// ---- POUs/Block/Cabines/Servomoteur_V1.TcPOU
FUNCTION_BLOCK Servomoteur_V1
VAR_INPUT
	Enable:					BOOL;	(*Mise en route du bloc de fonction*)
	Type_Consigne:			BOOL;	 (*Choix du type de pilotage du registre / 1 = ANA / 0 = TOR*)
	Mode_Vidange:			BOOL; 	(*Mode de vidange / 1=Mode vidange / 0= Mode alimentation douche, Douchette, Lavabo, etc...*)
	Cons_Pos_Dem:			REAL; 	(*Consigne position registre demandé (Venant de la régulation) / en %*)
	Cmd_Ouv_Dem:			BOOL; 	(*Commande ouverture registre demandé (Venant de la régulation) / 1 = Ouverture*)
	Info_Mes_Pos:			REAL; 	(*Info mesure position registre (recopie EAN) / en %*)
	Presence_Fdc:			INT; 	(*Mot de présence des fin de course / 0 = Pas de fin de course / 1 = Fin de course Ouvert / 2 = Fin de course Fermé / 3 = Les 2 fin de course*)
	Info_Fdc_Ouvert:			BOOL; 	(*Info fin de course ouvert (recopie ETOR) / 1 = Ouvert*)
	Info_Fdc_Ferme:			BOOL; 	(*Info fin de course fermé (recopi ETOR) / 1 = Fermé*)
	Secu_Niveau_Haut:		BOOL; 	(*Sécurité du niveau haut / 0 = Niveau haut actif*)
	Control_Discrodance:		BOOL;	 (*Autorisation de marche des alarmes / 1 = Alarme autorisé*)
	Hyst_Al_Discord:			REAL;	 (*Hystéresis pour le défaut discordance en type ANA*)
	Tempo_Discord_TOR:		TIME; 	(*Temporisation du défaut discordance en type TOR*)
	EF_Forcage:				BOOL;	 (*Enable forçage du registre / 1= Autorisé*)
	F_STOR_Registre: 		BOOL;	 (*Forçage du registre pour le mode TOR / 1= Forcé*)
	F_SAN_Registre:			REAL; 	(*Forçage du registre pour le mode ANA / en %*)
	Defaut_Alim_Eau:			BOOL;	(*Défaut sur l'alimentation d'eau*)
	E_Cmd_Rearmement:		BOOL;	(*Commande de réarmement*)
	In_SCL_In_MIN_REAL: REAL;
	In_SCL_In_MAX_REAL: REAL;
	In_SCL_Out_MIN_REAL: REAL;
	In_SCL_Out_MAX_REAL: REAL;
END_VAR
VAR_OUTPUT
	SAN_Cons_Registre:		INT; (*Consigne a appliqué au registre ANA (pour SAN) / en %*)
	STOR_Cmd_Ouv_Registre: BOOL; (*Commande a appliqué au registre TOR (pour STOR) / 1 = Ouverture*)
	Def_Discordance_ANA:BOOL;
	Def_Discordance_Ouverture:BOOL;
	Def_Discordance_Fermeture: BOOL;
END_VAR
VAR
	Cons_Registre:			REAL;
	iCons_Registre:			INT;
	Cmd_Registre:			BOOL;
	SCL_ANA: 				SCL;
	TON_1:					TON;
	TON_2:					TON;
	TON_3:					TON;
	TON_4:					TON;
	TON_5:					TON;
	TON_6:					TON;
	RS_1:					RS;
	RS_2:					RS;
	Calcul_1: REAL;
	Calcul_2: REAL;
END_VAR

IF(Enable)
	THEN
	(*======================Gestion de la Consigne===================================*)
	IF(Type_Consigne)
		THEN			(* Gestion consigne pour un registre ANA *)
		Cmd_Registre := FALSE;
		IF(EF_Forcage)
			THEN
				Cons_Registre := F_SAN_Registre;
			ELSE
				Cons_Registre := Cons_Pos_Dem;
		END_IF;
	ELSE				 (* Gestion consigne pour un registre TOR *)
		Cons_Registre := 0.0;
		IF(EF_Forcage)
			THEN
				Cmd_Registre := F_STOR_Registre;
			ELSE
				Cmd_Registre := Cmd_Ouv_Dem;
		END_IF
	END_IF;
	
	(*======================Gestion de la sortie Analogique==============================*)
	iCons_Registre := REAL_TO_INT(Cons_Registre); (*Convertion de la consigne analogique*)
	SCL_ANA(
		IN_INT:= iCons_Registre,
		LIM_MIN_IN_REAL:= In_SCL_In_MIN_REAL,
		LIM_MAX_IN_REAL:= In_SCL_In_MAX_REAL,
		LIM_MIN_OUT_REAL:= In_SCL_Out_MIN_REAL,(*0V*)
		LIM_MAX_OUT_REAL:= In_SCL_Out_MAX_REAL,(*10V*)
		OUT_INT=> SAN_Cons_Registre);
	
	(*======================Gestion de la sortie TOR====================================*)
	IF( Mode_Vidange)
		THEN (*Gestion de la STOR en fonction du mode de vidange*)
		IF(Secu_Niveau_Haut)
			THEN
				STOR_Cmd_Ouv_Registre := TRUE;
			ELSE
				STOR_Cmd_Ouv_Registre := Cmd_Registre;
		END_IF;
	ELSE (*Gestion de la STOR en fonction du mode alimentation*)
		IF(Secu_Niveau_Haut)
			THEN
				STOR_Cmd_Ouv_Registre := FALSE;
			ELSE
				STOR_Cmd_Ouv_Registre := Cmd_Registre AND NOT Defaut_Alim_Eau;
		END_IF;
	END_IF;
	
	(*======================Gestion du défaut de discordance============================*)
	IF(Control_Discrodance)
		THEN		(*Lors du contrôle de discordance*)
			IF(Type_Consigne)
				THEN		(* Alarme discordance pour registre SAN *)
					Calcul_1 := (Cons_Registre - Hyst_Al_Discord) ;
					Calcul_2 := (Cons_Registre + Hyst_Al_Discord) ;
					TON_1(IN := ((Calcul_1 > Info_Mes_Pos) OR (Calcul_2 < Info_Mes_Pos)),PT := Tempo_Discord_TOR);
					Def_Discordance_ANA:= TON_1.Q;
			ELSE			(* Alarme discordance pour registre STOR *)
				CASE Presence_Fdc OF
					0	:	(*Mode pas de fin de course*)
							Def_Discordance_Ouverture := FALSE;
							Def_Discordance_Fermeture := FALSE;
					1	:	(*Mode Fdc ouverture uniquement*)
							TON_2(IN := ( STOR_Cmd_Ouv_Registre AND NOT Info_Fdc_Ouvert ), PT := Tempo_Discord_TOR);
							Def_Discordance_Ouverture:= TON_2.Q;
							Def_Discordance_Fermeture := FALSE;
					2	:	(*Mode Fdc fermeture uniquement*)
							TON_3(IN := ( NOT STOR_Cmd_Ouv_Registre AND NOT Info_Fdc_Ferme ), PT := Tempo_Discord_TOR);
							Def_Discordance_Fermeture:= TON_3.Q;
							Def_Discordance_Ouverture := FALSE;
					3	:	(*Mode Fdc ouverture et fermeture*)
							TON_4(IN := ((STOR_Cmd_Ouv_Registre AND NOT Info_Fdc_Ouvert)),PT := Tempo_Discord_TOR);
							TON_5(IN := ((NOT STOR_Cmd_Ouv_Registre AND NOT Info_Fdc_Ferme )),PT := Tempo_Discord_TOR);
							TON_6(IN := (Info_Fdc_Ouvert AND Info_Fdc_Ferme) ,PT := Tempo_Discord_TOR);
							RS_1(SET:= TON_4.Q, RESET1:= Info_Fdc_Ouvert OR E_Cmd_Rearmement);
							RS_2(SET:= TON_5.Q, RESET1:= Info_Fdc_Ferme OR E_Cmd_Rearmement);
							Def_Discordance_Ouverture:= RS_1.Q1 OR TON_6.Q;
							Def_Discordance_Fermeture:= RS_2.Q1 OR TON_6.Q;
	
					ELSE  (*Si Presence_Fdc > à 3*)
					Def_Discordance_Ouverture := FALSE;
					Def_Discordance_Fermeture := FALSE;
				END_CASE;
			END_IF;
		ELSE		(* Si contrôle d'alarme discordance désactivé *)
			Def_Discordance_ANA := FALSE;
			Def_Discordance_Ouverture := FALSE;
			Def_Discordance_Fermeture := FALSE;
	END_IF;
	ELSE
			SAN_Cons_Registre := 0;
			STOR_Cmd_Ouv_Registre := FALSE;
			Def_Discordance_ANA := FALSE;
			Def_Discordance_Ouverture := FALSE;
			Def_Discordance_Fermeture := FALSE;
END_IF;

END_FUNCTION_BLOCK

// ---- POUs/p_Com_Modbus_RS485.TcPOU
PROGRAM p_Com_Modbus_RS485
VAR
	//Gestion de la com avec la passerelle LED
	Com_LED: Com485_Dalcnet;
	Lecture_Dimmer 	:INT;
	Lecture_Rouge 	:INT;
	Lecture_Vert 	:INT;
	Lecture_Bleu 	:INT;
	Lecture_Blanc 	:INT;
	LED_Com_Ok		:BOOL;
	LED_Com_Error	:BOOL;
	LED_Etape		:INT;
	
	//Gestion de la com avec GVL_RegTROX.Reg_Souf_GD_FCVT01
	FCVT01_Com_Ok		:BOOL;
	FCVT01_Com_Error	:BOOL;
	FCVT01_Etape		:INT;
	FCVT01_ConsAppli	:INT;
	
	//Gestion de la com avec GVL_RegTROX.Com_RegSouf_PD_FCVT02
	FCVT02_Com_Ok		:BOOL;
	FCVT02_Com_Error	:BOOL;
	FCVT02_Etape		:INT;
	FCVT02_ConsAppli	:INT;
	
	//Gestion de la com avec GVL_RegTROX.Com_RegSouf_Cabine_FCVT03
	FCVT03_Com_Ok		:BOOL;
	FCVT03_Com_Error	:BOOL;
	FCVT03_Etape		:INT;
	FCVT03_ConsAppli	:INT;
	
	//Gestion de la com avec GVL_RegTROX.Com_Reg_Bypass_FCVT04
	FCVT04_Com_Ok		:BOOL;
	FCVT04_Com_Error	:BOOL;
	FCVT04_Etape		:INT;
	FCVT04_ConsAppli	:INT;
	
	//Gestion de la com avec GVL_RegTROX.Com_RegSouf_CabGD_FCVT05
	FCVT05_Com_Ok		:BOOL;
	FCVT05_Com_Error	:BOOL;
	FCVT05_Etape		:INT;
	FCVT05_ConsAppli	:INT;
	
	//Gestion de la com avec GVL_RegTROX.Com_RegSouf_CabPD_FCVT06
	FCVT06_Com_Ok		:BOOL;
	FCVT06_Com_Error	:BOOL;
	FCVT06_Etape		:INT;
	FCVT06_ConsAppli	:INT;
	
	//Gestion de la com avec GVL_RegTROX.Com_RegRep_FCVT07
	FCVT07_Com_Ok		:BOOL;
	FCVT07_Com_Error	:BOOL;
	FCVT07_Etape		:INT;
	FCVT07_ConsAppli	:INT;
	
	Start_2: BOOL;
	Start_3: BOOL;
	Start_4: BOOL;
	Start_41: BOOL;
	Start_5: BOOL;
	Start_6: BOOL;
	Start_61: BOOL;
	Start_7: BOOL;
	Start_8: BOOL;
	Start_9: BOOL;
	FirstCycle: BOOL := TRUE;
	F_TRIG_0: F_TRIG;
	cpt: INT;
	CTU_Cpt: CTU;
	Cons_Cpt: WORD := 4;
	TOF_0: TOF;
	test: BOOL;
	
	//Gestion des forçages
	EF_FCVT01		:BOOL;
	F_FCVT01		:REAL;
	EF_FCVT02		:BOOL;
	F_FCVT02		:REAL;
	EF_FCVT03		:BOOL;
	F_FCVT03		:REAL;
	EF_FCVT04		:BOOL;
	F_FCVT04		:REAL;
	EF_FCVT05		:BOOL;
	F_FCVT05		:REAL;
	EF_FCVT06		:BOOL;
	F_FCVT06		:REAL;
	EF_FCVT07		:BOOL;
	F_FCVT07		:REAL;
END_VAR
VAR // added by the converter: edge detectors and wires of the graphical bodies
    _w1 : BOOL;
END_VAR

_w1 := Start_4 OR Start_6 OR Start_9;
Com_LED(
    Adresse_RS485 := 1,
    Start_Chenillard := _w1,
    In_Dimmer_Cabine := Cde_Dimmer_Cabine,
    In_Rouge_Cabine := Cde_Rouge_Cabine,
    In_Vert_Cabine := Cde_Vert_Cabine,
    In_Bleu_Cabine := Cde_Bleu_Cabine,
    In_Blanc_Cabine := Cde_Blanc_Cabine); // Com485_Dalcnet
LED_Com_Ok := Com_LED.Com_Ok;
LED_Com_Error := Com_LED.Com_Error;
LED_Etape := Com_LED.etape;
Defaut_Com_Dalcnet := Com_LED.Defaut_Com;
Lecture_Dimmer := Com_LED.Out_Dimmer_Cabine;
Lecture_Rouge := Com_LED.Out_Rouge_Cabine;
Lecture_Vert := Com_LED.Out_Vert_Cabine;
Lecture_Bleu := Com_LED.Out_Bleu_Cabine;
Lecture_Blanc := Com_LED.Out_Blanc_Cabine;
CTU_Cpt(CU := _w1, RESET := Start_8, PV := Cons_Cpt); // CTU
Cpt := CTU_Cpt.CV;
Start_2 := SEL(CTU_Cpt.CV = 1, false, Com_LED.Next_Chenillard);
Start_41 := SEL(CTU_Cpt.CV = 2, false, Com_LED.Next_Chenillard);
Start_61 := SEL(CTU_Cpt.CV = 3, false, Com_LED.Next_Chenillard);
GVL_RegTROX.Com_RegSouf_GD_FCVT01(
    Adresse_RS485 := 2,
    rEcriture_Cons_Deb := GVL_RegTROX.ConsAppliDeb_RegSouf_GD_FCVT01,
    rEcriture_Cons_Max := GVL_RegTROX.ConsMax_FCVT01,
    rEcriture_Cons_Min := GVL_RegTROX.ConsMin_FCVT01,
    Ecriture_ls_m3h := 1,
    Ecr_Interface_Mode := 1,
    Etat_Ma_Ventil := TRUE,
    TOL_Defaut_Discord := 250.0,
    Start_Chenillard := Start_2,
    EF_Forcage := EF_FCVT01,
    E_Forcage := F_FCVT01); // Com485_RegTROX
FCVT01_Com_Ok := GVL_RegTROX.Com_RegSouf_GD_FCVT01.Com_Ok;
FCVT01_Com_Error := GVL_RegTROX.Com_RegSouf_GD_FCVT01.Com_Error;
GVL_RegTROX.RegSouf_GD_FCVT01.Info_Mess_Pos := GVL_RegTROX.Com_RegSouf_GD_FCVT01.MES_Pos;
GVL_RegTROX.MES_RegSouf_GD_FCVT01.Mesure_EAN := GVL_RegTROX.Com_RegSouf_GD_FCVT01.rDebit_Relative;
FCVT01_ConsAppli := GVL_RegTROX.Com_RegSouf_GD_FCVT01.Lec_Cons_Appli;
FCVT01_Etape := GVL_RegTROX.Com_RegSouf_GD_FCVT01.etape;
GVL_RegTROX.RegSouf_GD_FCVT01_DefCom := GVL_RegTROX.Com_RegSouf_GD_FCVT01.Defaut_Com;
GVL_RegTROX.RegSouf_GD_FCVT01_Def_DiscordDeb := GVL_RegTROX.Com_RegSouf_GD_FCVT01.Defaut_Discord_Debit;
Start_3 := GVL_RegTROX.Com_RegSouf_GD_FCVT01.Next_Chenillard;
GVL_RegTROX.Com_RegSouf_PD_FCVT02(
    Adresse_RS485 := 3,
    rEcriture_Cons_Deb := GVL_RegTROX.ConsAppliDeb_RegSouf_PD_FCVT02,
    rEcriture_Cons_Max := GVL_RegTROX.ConsMax_FCVT02,
    rEcriture_Cons_Min := GVL_RegTROX.ConsMin_FCVT02,
    Ecriture_ls_m3h := 1,
    Ecr_Interface_Mode := 1,
    Etat_Ma_Ventil := TRUE,
    TOL_Defaut_Discord := 40.0,
    Start_Chenillard := Start_3,
    EF_Forcage := EF_FCVT02,
    E_Forcage := F_FCVT02); // Com485_RegTROX
FCVT02_Com_Ok := GVL_RegTROX.Com_RegSouf_PD_FCVT02.Com_Ok;
FCVT02_Com_Error := GVL_RegTROX.Com_RegSouf_PD_FCVT02.Com_Error;
GVL_RegTROX.RegSouf_PD_FCVT02.Info_Mess_Pos := GVL_RegTROX.Com_RegSouf_PD_FCVT02.MES_Pos;
GVL_RegTROX.MES_RegSouf_PD_FCVT02.Mesure_EAN := GVL_RegTROX.Com_RegSouf_PD_FCVT02.rDebit_Relative;
FCVT02_ConsAppli := GVL_RegTROX.Com_RegSouf_PD_FCVT02.Lec_Cons_Appli;
FCVT02_Etape := GVL_RegTROX.Com_RegSouf_PD_FCVT02.etape;
GVL_RegTROX.RegSouf_PD_FCVT02_DefCom := GVL_RegTROX.Com_RegSouf_PD_FCVT02.Defaut_Com;
GVL_RegTROX.RegSouf_PD_FCVT02_Def_DiscordDeb := GVL_RegTROX.Com_RegSouf_PD_FCVT02.Defaut_Discord_Debit;
Start_4 := GVL_RegTROX.Com_RegSouf_PD_FCVT02.Next_Chenillard;
GVL_RegTROX.Com_RegSouf_Cabine_FCVT03(
    Adresse_RS485 := 4,
    rEcriture_Cons_Deb := GVL_RegTROX.ConsAppliDeb_RegSouf_Cabine_FCVT03,
    rEcriture_Cons_Max := GVL_RegTROX.ConsMax_FCVT03,
    rEcriture_Cons_Min := GVL_RegTROX.ConsMin_FCVT03,
    Ecriture_ls_m3h := 1,
    Ecr_Interface_Mode := 1,
    Etat_Ma_Ventil := TRUE,
    TOL_Defaut_Discord := 1020.0,
    Start_Chenillard := Start_41,
    EF_Forcage := EF_FCVT03,
    E_Forcage := F_FCVT03); // Com485_RegTROX
FCVT03_Com_Ok := GVL_RegTROX.Com_RegSouf_Cabine_FCVT03.Com_Ok;
FCVT03_Com_Error := GVL_RegTROX.Com_RegSouf_Cabine_FCVT03.Com_Error;
GVL_RegTROX.RegSouf_Cabine_FCVT03.Info_Mess_Pos := GVL_RegTROX.Com_RegSouf_Cabine_FCVT03.MES_Pos;
GVL_RegTROX.MES_RegSouf_Cabine_FCVT03.Mesure_EAN := GVL_RegTROX.Com_RegSouf_Cabine_FCVT03.rDebit_Relative;
FCVT03_ConsAppli := GVL_RegTROX.Com_RegSouf_Cabine_FCVT03.Lec_Cons_Appli;
FCVT03_Etape := GVL_RegTROX.Com_RegSouf_Cabine_FCVT03.etape;
GVL_RegTROX.RegSouf_Cabine_FCVT03_DefCom := GVL_RegTROX.Com_RegSouf_Cabine_FCVT03.Defaut_Com;
GVL_RegTROX.RegSouf_Cabine_FCVT03_Def_DiscordDeb := GVL_RegTROX.Com_RegSouf_Cabine_FCVT03.Defaut_Discord_Debit;
Start_5 := GVL_RegTROX.Com_RegSouf_Cabine_FCVT03.Next_Chenillard;
GVL_RegTROX.Com_Reg_Bypass_FCVT04(
    Adresse_RS485 := 5,
    rEcriture_Cons_Deb := GVL_RegTROX.ConsAppliDeb_Reg_Bypass_FCVT04,
    rEcriture_Cons_Max := GVL_RegTROX.ConsMax_FCVT04,
    rEcriture_Cons_Min := GVL_RegTROX.ConsMin_FCVT04,
    Ecriture_ls_m3h := 1,
    Ecr_Interface_Mode := 1,
    Etat_Ma_Ventil := TRUE,
    TOL_Defaut_Discord := 150.0,
    Start_Chenillard := Start_5,
    EF_Forcage := EF_FCVT04,
    E_Forcage := F_FCVT04); // Com485_RegTROX
FCVT04_Com_Ok := GVL_RegTROX.Com_Reg_Bypass_FCVT04.Com_Ok;
FCVT04_Com_Error := GVL_RegTROX.Com_Reg_Bypass_FCVT04.Com_Error;
GVL_RegTROX.RegBypass_FCVT04.Info_Mess_Pos := GVL_RegTROX.Com_Reg_Bypass_FCVT04.MES_Pos;
GVL_RegTROX.MES_RegBypass_FCVT04.Mesure_EAN := GVL_RegTROX.Com_Reg_Bypass_FCVT04.rDebit_Relative;
FCVT04_ConsAppli := GVL_RegTROX.Com_Reg_Bypass_FCVT04.Lec_Cons_Appli;
FCVT04_Etape := GVL_RegTROX.Com_Reg_Bypass_FCVT04.etape;
GVL_RegTROX.Reg_Bypass_FCVT04_DefCom := GVL_RegTROX.Com_Reg_Bypass_FCVT04.Defaut_Com;
GVL_RegTROX.Reg_Bypass_FCVT04_Def_DiscordDeb := GVL_RegTROX.Com_Reg_Bypass_FCVT04.Defaut_Discord_Debit;
Start_6 := GVL_RegTROX.Com_Reg_Bypass_FCVT04.Next_Chenillard;
GVL_RegTROX.Com_RegSouf_CabGD_FCVT05(
    Adresse_RS485 := 6,
    rEcriture_Cons_Deb := GVL_RegTROX.ConsAppliDeb_RegSouf_CabGD_FCVT05,
    rEcriture_Cons_Max := GVL_RegTROX.ConsMax_FCVT05,
    rEcriture_Cons_Min := GVL_RegTROX.ConsMin_FCVT05,
    Ecriture_ls_m3h := 1,
    Ecr_Interface_Mode := 1,
    Etat_Ma_Ventil := TRUE,
    TOL_Defaut_Discord := 250.0,
    Start_Chenillard := Start_61,
    EF_Forcage := EF_FCVT05,
    E_Forcage := F_FCVT05); // Com485_RegTROX
FCVT05_Com_Ok := GVL_RegTROX.Com_RegSouf_CabGD_FCVT05.Com_Ok;
FCVT05_Com_Error := GVL_RegTROX.Com_RegSouf_CabGD_FCVT05.Com_Error;
GVL_RegTROX.RegSouf_CabGD_FCVT05.Info_Mess_Pos := GVL_RegTROX.Com_RegSouf_CabGD_FCVT05.MES_Pos;
GVL_RegTROX.MES_RegSouf_CabGD_FCVT05.Mesure_EAN := GVL_RegTROX.Com_RegSouf_CabGD_FCVT05.rDebit_Relative;
FCVT05_ConsAppli := GVL_RegTROX.Com_RegSouf_CabGD_FCVT05.Lec_Cons_Appli;
FCVT05_Etape := GVL_RegTROX.Com_RegSouf_CabGD_FCVT05.etape;
GVL_RegTROX.RegSouf_CabGD_FCVT05_DefCom := GVL_RegTROX.Com_RegSouf_CabGD_FCVT05.Defaut_Com;
GVL_RegTROX.RegSouf_CabGD_FCVT05_Def_DiscordDeb := GVL_RegTROX.Com_RegSouf_CabGD_FCVT05.Defaut_Discord_Debit;
Start_7 := GVL_RegTROX.Com_RegSouf_CabGD_FCVT05.Next_Chenillard;
GVL_RegTROX.Com_RegSouf_CabPD_FCVT06(
    Adresse_RS485 := 7,
    rEcriture_Cons_Deb := GVL_RegTROX.ConsAppliDeb_RegSouf_CabPD_FCVT06,
    rEcriture_Cons_Max := GVL_RegTROX.ConsMax_FCVT06,
    rEcriture_Cons_Min := GVL_RegTROX.ConsMin_FCVT06,
    Ecriture_ls_m3h := 1,
    Ecr_Interface_Mode := 1,
    Etat_Ma_Ventil := TRUE,
    TOL_Defaut_Discord := 50.0,
    Start_Chenillard := Start_7,
    EF_Forcage := EF_FCVT06,
    E_Forcage := F_FCVT06); // Com485_RegTROX
FCVT06_Com_Ok := GVL_RegTROX.Com_RegSouf_CabPD_FCVT06.Com_Ok;
FCVT06_Com_Error := GVL_RegTROX.Com_RegSouf_CabPD_FCVT06.Com_Error;
GVL_RegTROX.RegSouf_CabPD_FCVT06.Info_Mess_Pos := GVL_RegTROX.Com_RegSouf_CabPD_FCVT06.MES_Pos;
GVL_RegTROX.MES_RegSouf_CabPD_FCVT06.Mesure_EAN := GVL_RegTROX.Com_RegSouf_CabPD_FCVT06.rDebit_Relative;
FCVT06_ConsAppli := GVL_RegTROX.Com_RegSouf_CabPD_FCVT06.Lec_Cons_Appli;
FCVT06_Etape := GVL_RegTROX.Com_RegSouf_CabPD_FCVT06.etape;
GVL_RegTROX.RegSouf_CabPD_FCVT06_DefCom := GVL_RegTROX.Com_RegSouf_CabPD_FCVT06.Defaut_Com;
GVL_RegTROX.RegSouf_CabPD_FCVT06_Def_DiscordDeb := GVL_RegTROX.Com_RegSouf_CabPD_FCVT06.Defaut_Discord_Debit;
Start_8 := GVL_RegTROX.Com_RegSouf_CabPD_FCVT06.Next_Chenillard;
GVL_RegTROX.Com_RegRep_FCVT07(
    Adresse_RS485 := 8,
    rEcriture_Cons_Deb := GVL_RegTROX.ConsAppliDeb_RegRep_FCVT07,
    rEcriture_Cons_Max := GVL_RegTROX.ConsMax_FCVT07,
    rEcriture_Cons_Min := GVL_RegTROX.ConsMin_FCVT07,
    Ecriture_ls_m3h := 1,
    Ecr_Interface_Mode := 1,
    Etat_Ma_Ventil := TRUE,
    TOL_Defaut_Discord := 1020.0,
    Start_Chenillard := Start_8,
    EF_Forcage := EF_FCVT07,
    E_Forcage := F_FCVT07); // Com485_RegTROX
FCVT07_Com_Ok := GVL_RegTROX.Com_RegRep_FCVT07.Com_Ok;
FCVT07_Com_Error := GVL_RegTROX.Com_RegRep_FCVT07.Com_Error;
GVL_RegTROX.RegRep_FCVT07.Info_Mess_Pos := GVL_RegTROX.Com_RegRep_FCVT07.MES_Pos;
GVL_RegTROX.MES_RegRep_FCVT07.Mesure_EAN := GVL_RegTROX.Com_RegRep_FCVT07.rDebit_Relative;
FCVT07_ConsAppli := GVL_RegTROX.Com_RegRep_FCVT07.Lec_Cons_Appli;
FCVT07_Etape := GVL_RegTROX.Com_RegRep_FCVT07.etape;
GVL_RegTROX.RegRep_FCVT07_DefCom := GVL_RegTROX.Com_RegRep_FCVT07.Defaut_Com;
GVL_RegTROX.RegRep_FCVT07_Def_DiscordDeb := GVL_RegTROX.Com_RegRep_FCVT07.Defaut_Discord_Debit;
F_TRIG_0(CLK := FirstCycle OR test); // F_TRIG
Start_9 := GVL_RegTROX.Com_RegRep_FCVT07.Next_Chenillard OR F_TRIG_0.Q;
TOF_0(IN := Start_2, PT := T#5m); // TOF
test := TOF_0.Q;
FirstCycle := FALSE;

END_PROGRAM

// ---- POUs/Block/Cabines/Com485_Dalcnet.TcPOU
FUNCTION_BLOCK Com485_Dalcnet
VAR_INPUT
	Adresse_RS485		:BYTE;
	Start_Chenillard	: BOOL;
	In_Dimmer_Cabine	:INT;
	In_Rouge_Cabine		:INT;
	In_Vert_Cabine		:INT;
	In_Bleu_Cabine		:INT;
	In_Blanc_Cabine		:INT;
END_VAR
VAR_OUTPUT
	Com_Ok 				: BOOL;
	Com_Error 			: BOOL;
	etape				: INT := 0;
	Defaut_Com			: BOOL;
	Next_Chenillard		: BOOL;
	Out_Dimmer_Cabine	:INT;
	Out_Rouge_Cabine	:INT;
	Out_Vert_Cabine		:INT;
	Out_Bleu_Cabine		:INT;
	Out_Blanc_Cabine	:INT;
END_VAR
VAR
	Last_Error				: MODBUS_ERRORS;
	ValeursEcrites_Dalcnet 	: ARRAY[0..5] OF INT;
	ValeursLues_Dalcnet 	: ARRAY[0..5] OF INT;
	Chgt_Ecr_Cons_Dalcnet	: BOOL;
	F_TRIG_1				: F_TRIG;
	F_TRIG_2				: F_TRIG;
	TON_1					: TON;
	TON_2					: TON;
	R_TRIG_Start			: R_TRIG;
END_VAR

(*Gestion de l'ecriture*)
ValeursEcrites_Dalcnet[0] 	:= In_Dimmer_Cabine;
ValeursEcrites_Dalcnet[1] 	:= In_Rouge_Cabine;
ValeursEcrites_Dalcnet[2] 	:= In_Vert_Cabine;
ValeursEcrites_Dalcnet[3] 	:= In_Bleu_Cabine;
ValeursEcrites_Dalcnet[4] 	:= In_Blanc_Cabine;
(*Recopie des consignes du Dalcnet*)
Out_Dimmer_Cabine 			:= ValeursLues_Dalcnet[0];
Out_Rouge_Cabine 			:= ValeursLues_Dalcnet[1];
Out_Vert_Cabine 			:= ValeursLues_Dalcnet[2];
Out_Bleu_Cabine 			:= ValeursLues_Dalcnet[3];
Out_Blanc_Cabine 			:= ValeursLues_Dalcnet[4];

(*Changement de consigne pour l'ecriture Modbus*)
IF((Out_Rouge_Cabine <> In_Rouge_Cabine) OR (Out_Vert_Cabine <> In_Vert_Cabine) OR (Out_Bleu_Cabine <> In_Bleu_Cabine) OR (Out_Blanc_Cabine <> In_Blanc_Cabine))
	THEN
	Chgt_Ecr_Cons_Dalcnet := TRUE;
	ELSE
	Chgt_Ecr_Cons_Dalcnet := FALSE;
END_IF;

(**********************************************Gestion sécurité anti-blocage*)
(*En cas de blocage de la variable etape à 0*)
TON_1(IN:=(etape = 1) , PT:= T#3S);
IF (TON_1.Q) THEN etape := 3; END_IF;

(*En cas de blocage de la variable etape à 3*)
TON_2(IN:=(etape = 3) , PT:= T#3S);
IF (TON_2.Q) THEN etape := 0; END_IF;

(**********************************************Lecture/ecriture modbus*)
CASE etape OF
	0: (*Etape Attente*)
		R_TRIG_Start(CLK:= Start_Chenillard);
		IF (R_TRIG_Start.Q)
			THEN
			etape := etape + 1;
		END_IF;
		Next_Chenillard := FALSE;
	(*Lecture dalcnet*)
	1:	MB.ReadRegs(	Execute := NOT MB.BUSY,
						UnitID := Adresse_RS485,
						Quantity := 6,								(* Lecture de 6 mots *)
						MBAddr := 16#0,							(*A partir de l'adresse 0*)
						cbLength := SIZEOF(ValeursLues_Dalcnet),
						pMemoryAddr := ADR(ValeursLues_Dalcnet),
						Timeout := T#5000MS);
		F_TRIG_1(CLK:= MB.BUSY);
		IF(F_TRIG_1.Q)
			THEN
			etape := etape + 1;
		END_IF;
	2:	IF MB.Error THEN
			Com_Ok := FALSE;
			Com_Error := TRUE;
			Last_Error := MB.ErrorId;
		ELSE
			Com_Ok := TRUE;
			Com_Error := FALSE;
			Last_Error := 0;
		END_IF
		etape := etape + 1;

		(*Ecriture dalcnet*)
	3:	MB.WriteRegs(	Execute := (NOT MB.BUSY AND Chgt_Ecr_Cons_Dalcnet),
						UnitID := Adresse_RS485,
						Quantity := 6,								(* Ecriture de 6 mots *)
						MBAddr := 16#0,							(*A partir de l'adresse 0*)
						cbLength := SIZEOF(ValeursEcrites_Dalcnet),
						pMemoryAddr := ADR(ValeursEcrites_Dalcnet),
						Timeout := T#5000ms);
		F_TRIG_2(CLK:= MB.BUSY);
		Next_Chenillard := TRUE;
		IF(F_TRIG_2.Q OR NOT Chgt_Ecr_Cons_Dalcnet)
			THEN
			etape := etape + 1;
		END_IF;
	4:	IF MB.Error THEN
			Com_Ok := FALSE;
			Com_Error := TRUE;
			Last_Error := MB.ErrorId;
		ELSE
			Com_Ok := TRUE;
			Com_Error := FALSE;
			Last_Error := 0;
		END_IF
		etape := 0;
END_CASE;

END_FUNCTION_BLOCK

// ---- POUs/Block/Cabines/Com485_RegTROX.TcPOU
FUNCTION_BLOCK Com485_RegTROX
VAR_INPUT
	Adresse_RS485		:BYTE;
	rEcriture_Cons_Deb	: REAL;
	rEcriture_Cons_Max 	: REAL;
	rEcriture_Cons_Min 	: REAL;
	Ecriture_ls_m3h		: INT := 1; (*(0=l/s - 1=m3/h - 6 =cfm)*)
	Ecr_Interface_Mode	: INT := 1; (*0=Consigne via 0-10V / 1=Consigne via Modbus*)
	Etat_Ma_Ventil		: BOOL;
	TOL_Defaut_Discord	: REAL;
	Start_Chenillard	: BOOL;
	EF_Forcage			: BOOL;
	E_Forcage			: REAL;
END_VAR
VAR_OUTPUT
	Com_Ok 				: BOOL;
	Com_Error 			: BOOL;
	MES_Pos				: REAL;
	rDebit_Relative 	: REAL;
	Lec_Cons_Appli		: INT;
	Lecture_Cons_Max 	: INT;
	Lecture_Cons_Min 	: INT;
	Lecture_ls_m3h 		: INT; (*(0=l/s - 1=m3/h - 6 =cfm)*)
	Lec_Interface_Mode	: INT; (*0=Consigne via 0-10V / 1=Consigne via Modbus*)
	etape				: INT := 0;
	Defaut_Com			: BOOL;
	Defaut_Discord_Debit	: BOOL;
	Next_Chenillard		: BOOL;
END_VAR
VAR
	Last_Error			: MODBUS_ERRORS;
	ValeursLues1 		:ARRAY[1..4] OF INT;
	ValeursLues2 		:ARRAY[1..2] OF INT;
	ValeursLues3  		:ARRAY[1..3] OF INT;
	Posi_Relative 		: INT;
	Posi_Absolue		 :INT;
	Debit_Absolue 		: INT;
	Lecture_Etat 			: INT;
	Lecture_Adresse 		: INT;
	Lecture_Software 		: INT;
	
	Ecriture_Cons_Deb	: INT;
	Ecriture_Cons_Max 	: INT;
	Ecriture_Cons_Min 	: INT;
	Debit_Relative 		: INT;

	Changement_Ecr_Cons: BOOL;
	Changement_Ecr_Interface_Mode : BOOL;
	Changement_Ecr_ls_m3h : BOOL;
	Changement_Ecr_Cons_Min : BOOL;
	Changement_Ecr_Cons_Max : BOOL;
	
(*Gestion du registre de soufflage*)
	F_TRIG_3: F_TRIG;
	F_TRIG_4: F_TRIG;
	F_TRIG_5: F_TRIG;
	F_TRIG_6: F_TRIG;
	F_TRIG_7: F_TRIG;
	F_TRIG_8: F_TRIG;
	F_TRIG_9: F_TRIG;
	F_TRIG_10: F_TRIG;
	F_TRIG_11: F_TRIG;
	F_TRIG_12: F_TRIG;		
	F_TRIG_13: F_TRIG;

(*Autres*)
	TON_1: TON;
	TON_2: TON;
	TON_3: TON;
	TON_4: TON;
	TON_5: TON;
	TON_6: TON;
	TON_7: TON;
	TON_8: TON;
	TON_9: TON;
	TON_10: TON;
	TON_11: TON;

(********Gestion des défauts de communication*)
	TON_Com :TON;
	RS_Def_Com: RS;

(********Gestion des défauts de discrodance du débit*)
	Var_ABS_Debit		:REAL;
	TON_DefDiscord		:TON;
	R_TRIG_Start: R_TRIG;
END_VAR

// Gestion du forçage de la consigne
IF (EF_Forcage) THEN
	rEcriture_Cons_Deb := E_Forcage;
	ELSE
	rEcriture_Cons_Deb := rEcriture_Cons_Deb;
END_IF

// Conversion des variables
Ecriture_Cons_Deb := REAL_TO_INT(rEcriture_Cons_Deb);
Ecriture_Cons_Max := REAL_TO_INT(rEcriture_Cons_Max);
Ecriture_Cons_Min := REAL_TO_INT(rEcriture_Cons_Min);
rDebit_Relative := INT_TO_REAL(Debit_Relative);

(**********************************************Gestion de la communication avec le registre d'extraction numéro 7*)
(*Information ouverture du registre*)
Posi_Relative := ValeursLues1[1];
(*Mesure du débit du registre*)
Debit_Relative := ValeursLues1[4];
Lec_Cons_Appli := Lec_Cons_Appli;
MES_Pos := Posi_Relative / 100.0; (*Récupération de la valeur de position du registre de soufflage*)
(*Information des consignes Min/Max applicable au registre*)
Lecture_Cons_Max := ValeursLues3[2];
Lecture_Cons_Min := ValeursLues3[1];
(*Information d'état de l'unité de lecture du débit (0=l/s - 1=m3/h - 6 =cfm)*)
Lecture_ls_m3h := Lecture_ls_m3h;
(*Autres informations*)
Posi_Absolue := ValeursLues1[2];
Debit_Absolue := ValeursLues1[3];
Lecture_Etat := ValeursLues2[2];
Lecture_Adresse := Lecture_Adresse;
Lecture_Software := ValeursLues2[1];
Lec_Interface_Mode := ValeursLues3[3]; (*0=Consigne via 0-10V / 1=Consigne via Modbus*)

(*Changement de consigne pour l'ecriture Modbus*)
IF((Lec_Cons_Appli <> Ecriture_Cons_Deb))
	THEN
	Changement_Ecr_Cons := TRUE;
	ELSE
	Changement_Ecr_Cons := FALSE;
END_IF;

(*Changement de l'ecriture interface mode*)
IF((Lec_Interface_Mode <> Ecr_Interface_Mode))
	THEN
	Changement_Ecr_Interface_Mode := TRUE;
	ELSE
	Changement_Ecr_Interface_Mode := FALSE;
END_IF;

(*Changement de l'ecriture de l'unité du débit*)
IF((Lecture_ls_m3h <> Ecriture_ls_m3h))
	THEN
	Changement_Ecr_ls_m3h := TRUE;
	ELSE
	Changement_Ecr_ls_m3h := FALSE;
END_IF;

(*Changement de l'ecriture de la consigne minimmum*)
IF((Lecture_Cons_Min <> Ecriture_Cons_Min))
	THEN
	Changement_Ecr_Cons_Min := TRUE;
	ELSE
	Changement_Ecr_Cons_Min := FALSE;
END_IF;

(*Changement de l'ecriture de la consigne maximum*)
IF((Lecture_Cons_Max <> Ecriture_Cons_Max))
	THEN
	Changement_Ecr_Cons_Max := TRUE;
	ELSE
	Changement_Ecr_Cons_Max := FALSE;
END_IF;

(**********************************************Gestion sécurité anti-blocage*)
(*En cas de blocage de la variable etape à 1*)
TON_1(IN:=(etape = 1) , PT:= T#3s);
IF (TON_1.Q) THEN etape := 3; END_IF;

(*En cas de blocage de la variable etape à 3*)
TON_2(IN:=(etape = 3) , PT:= T#3s);
IF (TON_2.Q) THEN etape := 5; END_IF;

(*En cas de blocage de la variable etape à 5*)
TON_3(IN:=(etape = 5) , PT:= T#3s);
IF (TON_3.Q) THEN etape := 7; END_IF;

(*En cas de blocage de la variable etape à 7*)
TON_4(IN:=(etape = 7) , PT:= T#3s);
IF (TON_4.Q) THEN etape := 9; END_IF;

(*En cas de blocage de la variable etape à 9*)
TON_5(IN:=(etape = 9) , PT:= T#3s);
IF (TON_5.Q) THEN etape := 11; END_IF;

(*En cas de blocage de la variable etape à 11*)
TON_6(IN:=(etape = 11) , PT:= T#3s);
IF (TON_6.Q) THEN etape := 13; END_IF;

(*En cas de blocage de la variable etape à 13*)
TON_7(IN:=(etape = 13) , PT:= T#3s);
IF (TON_7.Q) THEN etape := 15; END_IF;

(*En cas de blocage de la variable etape à 15*)
TON_8(IN:=(etape = 15) , PT:= T#3s);
IF (TON_8.Q) THEN etape := 17; END_IF;

(*En cas de blocage de la variable etape à 17*)
TON_9(IN:=(etape = 17) , PT:= T#3s);
IF (TON_9.Q) THEN etape := 19; END_IF;

(*En cas de blocage de la variable etape à 19*)
TON_10(IN:=(etape = 19) , PT:= T#3s);
IF (TON_10.Q) THEN etape := 21; END_IF;

(*En cas de blocage de la variable etape à 21*)
TON_11(IN:=(etape = 21) , PT:= T#3s);
IF (TON_11.Q) THEN etape := 0; END_IF;

CASE etape OF
	0: (*Etape Attente*)
		R_TRIG_Start(CLK:= Start_Chenillard);
		IF (R_TRIG_Start.Q)
			THEN
			etape := etape + 1;
		END_IF;
		Next_Chenillard := FALSE;
	(* Lecture Registre ultrason soufflage*)
	1:	MB.ReadRegs(	Execute := NOT MB.BUSY,
						UnitID := Adresse_RS485,
						Quantity := 4,								(* Lecture de 4 mots *)
						MBAddr := 16#4,							(*A partir de l'adresse 4*)
						cbLength := SIZEOF(ValeursLues1),
						pMemoryAddr := ADR(ValeursLues1),
						Timeout := T#1000ms);
		F_TRIG_3(CLK:= MB.BUSY);
		IF(F_TRIG_3.Q)
			THEN
			etape := etape + 1;
		END_IF;
	2:	IF MB.Error THEN
			Com_Ok := FALSE;
			Com_Error := TRUE;
			Last_Error := MB.ErrorId;
		ELSE
			Com_Ok := TRUE;
			Com_Error := FALSE;
			Last_Error := 0;
		END_IF
		etape := etape + 1;

	3:	MB.ReadRegs(	Execute := (NOT MB.BUSY),
						UnitID := Adresse_RS485,
						Quantity := 2,								(* Lecture de 2 mots *)
						MBAddr := 16#67,							(*A partir de l'adresse 103*)
						cbLength := SIZEOF(ValeursLues2),
						pMemoryAddr := ADR(ValeursLues2),
						Timeout := T#1000ms);
		F_TRIG_4(CLK:= MB.BUSY);
		IF(F_TRIG_4.Q)
			THEN
			etape := etape + 1;
		END_IF;
	4:	IF MB.Error THEN
			Com_Ok := FALSE;
			Com_Error := TRUE;
			Last_Error := MB.ErrorId;
		ELSE
			Com_Ok := TRUE;
			Com_Error := FALSE;
			Last_Error := 0;
		END_IF
		etape := etape + 1;

	5:	MB.ReadRegs(	Execute := (NOT MB.BUSY),
						UnitID := Adresse_RS485,
						Quantity := 3,								(* Lecture de 3 mots *)
						MBAddr := 16#78,							(*A partir de l'adresse 120*)
						cbLength := SIZEOF(ValeursLues3),
						pMemoryAddr := ADR(ValeursLues3),
						Timeout := T#1000ms);
		F_TRIG_5(CLK:= MB.BUSY);
		IF(F_TRIG_5.Q)
			THEN
			etape := etape + 1;
		END_IF;
	6:	IF MB.Error THEN
			Com_Ok := FALSE;
			Com_Error := TRUE;
			Last_Error := MB.ErrorId;
		ELSE
			Com_Ok := TRUE;
			Com_Error := FALSE;
			Last_Error := 0;
		END_IF
		etape := etape + 1;

	7:	MB.ReadRegs(	Execute := (NOT MB.BUSY),
						UnitID := Adresse_RS485,
						Quantity := 1,								(* Lecture de 1 mots *)
						MBAddr := 16#82,							(*A partir de l'adresse 130*)
						cbLength := SIZEOF(Lecture_Adresse),
						pMemoryAddr := ADR(Lecture_Adresse),
						Timeout := T#1000ms);
		F_TRIG_6(CLK:= MB.BUSY);
		IF(F_TRIG_6.Q)
			THEN
			etape := etape + 1;
		END_IF;
	8:	IF MB.Error THEN
			Com_Ok := FALSE;
			Com_Error := TRUE;
			Last_Error := MB.ErrorId;
		ELSE
			Com_Ok := TRUE;
			Com_Error := FALSE;
			Last_Error := 0;
		END_IF
		etape := etape + 1;

	9:	MB.ReadRegs(	Execute := (NOT MB.BUSY),
						UnitID := Adresse_RS485,
						Quantity := 1,								(* Lecture de 1 mots *)
						MBAddr := 16#C9,							(*A partir de l'adresse 201*)
						cbLength := SIZEOF(Lecture_ls_m3h),
						pMemoryAddr := ADR(Lecture_ls_m3h),
						Timeout := T#1000ms);
		F_TRIG_7(CLK:= MB.BUSY);
		IF(F_TRIG_7.Q)
			THEN
			etape := etape + 1;
		END_IF;
	10:	IF MB.Error THEN
			Com_Ok := FALSE;
			Com_Error := TRUE;
			Last_Error := MB.ErrorId;
		ELSE
			Com_Ok := TRUE;
			Com_Error := FALSE;
			Last_Error := 0;
		END_IF
		etape := etape + 1;

	11:	MB.WriteSingleRegister(	Execute := (NOT MB.BUSY AND Changement_Ecr_Cons_Min),
						UnitID := Adresse_RS485,
						Quantity := 1,								(* Ecriture de 1 mots *)
						MBAddr := 16#78,							(*A partir de l'adresse 120*)
						cbLength := SIZEOF(Ecriture_Cons_Min),
						pMemoryAddr := ADR(Ecriture_Cons_Min),
						Timeout := T#1000ms);
		F_TRIG_8(CLK:= MB.BUSY);
		IF(F_TRIG_8.Q OR NOT Changement_Ecr_Cons_Min)
			THEN
			etape := etape + 1;
		END_IF;
	12:	IF MB.Error THEN
			Com_Ok := FALSE;
			Com_Error := TRUE;
			Last_Error := MB.ErrorId;
		ELSE
			Com_Ok := TRUE;
			Com_Error := FALSE;
			Last_Error := 0;
		END_IF
		etape := etape + 1;

	13:	MB.WriteSingleRegister(	Execute := (NOT MB.BUSY AND Changement_Ecr_Cons_Max),
						UnitID := Adresse_RS485,
						Quantity := 1,								(* Ecriture de 1 mots *)
						MBAddr := 16#79,							(*A partir de l'adresse 121*)
						cbLength := SIZEOF(Ecriture_Cons_Max),
						pMemoryAddr := ADR(Ecriture_Cons_Max),
						Timeout := T#1000ms);
		F_TRIG_9(CLK:= MB.BUSY);
		IF(F_TRIG_9.Q OR NOT Changement_Ecr_Cons_Max)
			THEN
			etape := etape + 1;
		END_IF;
	14:	IF MB.Error THEN
			Com_Ok := FALSE;
			Com_Error := TRUE;
			Last_Error := MB.ErrorId;
		ELSE
			Com_Ok := TRUE;
			Com_Error := FALSE;
			Last_Error := 0;
		END_IF
		etape := etape + 1;

	15:	MB.WriteSingleRegister(	Execute := (NOT MB.BUSY  AND Changement_Ecr_ls_m3h),
						UnitID := Adresse_RS485,
						Quantity := 1,								(* Ecriture de 1 mots *)
						MBAddr := 16#C9,							(*A partir de l'adresse 201*)
						cbLength := SIZEOF(Ecriture_ls_m3h),
						pMemoryAddr := ADR(Ecriture_ls_m3h),
						Timeout := T#1000ms);
		F_TRIG_10(CLK:= MB.BUSY);
		IF(F_TRIG_10.Q OR NOT Changement_Ecr_ls_m3h)
			THEN
			etape := etape + 1;
		END_IF;
	16:	IF MB.Error THEN
			Com_Ok := FALSE;
			Com_Error := TRUE;
			Last_Error := MB.ErrorId;
		ELSE
			Com_Ok := TRUE;
			Com_Error := FALSE;
			Last_Error := 0;
		END_IF
		etape := etape + 1;
		
	17:	MB.ReadRegs(	Execute := (NOT MB.BUSY),
						UnitID := Adresse_RS485,
						Quantity := 1,								(* Lecture de 1 mots *)
						MBAddr := 16#14,							(*A partir de l'adresse 20*)
						cbLength := SIZEOF(Lec_Cons_Appli),
						pMemoryAddr := ADR(Lec_Cons_Appli),
						Timeout := T#1000ms);
		F_TRIG_11(CLK:= MB.BUSY);
		IF(F_TRIG_11.Q)
			THEN
			etape := etape + 1;
		END_IF;
	18:	IF MB.Error THEN
			Com_Ok := FALSE;
			Com_Error := TRUE;
			Last_Error := MB.ErrorId;
		ELSE
			Com_Ok := TRUE;
			Com_Error := FALSE;
			Last_Error := 0;
		END_IF
		etape := etape + 1;
	
	19:	MB.WriteSingleRegister(	Execute := (NOT MB.BUSY AND Changement_Ecr_Cons),
						UnitID := Adresse_RS485,
						Quantity := 1,								(* Ecriture de 1 mots *)
						MBAddr := 16#14,							(*A partir de l'adresse 20*)
						cbLength := SIZEOF(Ecriture_Cons_Deb),
						pMemoryAddr := ADR(Ecriture_Cons_Deb),
						Timeout := T#1000ms);
		F_TRIG_12(CLK:= MB.BUSY);
		IF(F_TRIG_12.Q OR NOT Changement_Ecr_Cons)
			THEN
			etape := etape + 1;
		END_IF;
	20:	IF MB.Error THEN
			Com_Ok := FALSE;
			Com_Error := TRUE;
			Last_Error := MB.ErrorId;
		ELSE
			Com_Ok := TRUE;
			Com_Error := FALSE;
			Last_Error := 0;
		END_IF
		etape := etape + 1;

	21:	MB.WriteSingleRegister(	Execute := (NOT MB.BUSY AND Changement_Ecr_Interface_Mode),
						UnitID := Adresse_RS485,
						Quantity := 1,								(* Ecriture de 1 mots *)
						MBAddr := 16#7A,							(*A partir de l'adresse 122*)
						cbLength := SIZEOF(Ecr_Interface_Mode),
						pMemoryAddr := ADR(Ecr_Interface_Mode),
						Timeout := T#1000ms);
		F_TRIG_13(CLK:= MB.BUSY);
		IF(F_TRIG_13.Q OR NOT Changement_Ecr_Interface_Mode)
			THEN
			etape := etape + 1;
		END_IF;
	22:	IF MB.Error THEN
			Com_Ok := FALSE;
			Com_Error := TRUE;
			Last_Error := MB.ErrorId;
		ELSE
			Com_Ok := TRUE;
			Com_Error := FALSE;
			Last_Error := 0;
		END_IF
		Next_Chenillard := TRUE;
		etape := 0;
END_CASE

(**********************************************Gestion des défauts de communication*)
TON_Com(IN:= (Com_Ok) , PT:= t#4s );
RS_Def_Com(		SET:= (Com_Error),
				RESET1:= (TON_Com.Q));
Defaut_Com := RS_Def_Com.Q1;

(**********************************************gestion défaut discordance de la mesure de débit*)
Var_ABS_Debit := ABS(Lec_Cons_Appli - Debit_Relative);
TON_DefDiscord(IN:= (Var_ABS_Debit > TOL_Defaut_Discord) AND Etat_Ma_Ventil, PT:= t#3600s);
IF(TON_DefDiscord.Q)
	THEN
	Defaut_Discord_Debit := TRUE;
	ELSE
	Defaut_Discord_Debit := FALSE;
END_IF;

END_FUNCTION_BLOCK

// ---- POUs/Block/Objets/Objet_Registre_V1.TcPOU
FUNCTION_BLOCK Objet_Registre_V1
VAR_INPUT
	Cons_Pos_Dem		:REAL;	(*Consigne position registre demandé (Venant de la Régulation) / en %*)
	Cmd_Ouv_Dem		:BOOL;	(*Commande ouverture registre demandé (Venant de la Régulation) / 1 = Ouverture*)
	Info_Mess_Pos		:REAL;	(*nfo mesure position registre (recopie EAN) / en %*)
	Info_Fdc_ouvert		:BOOL;	(*Info fin de course ouvert (recopie ETOR) / 1 = Ouvert*)
	Info_Fdc_ferme		:BOOL;	(*Info fin de course fermé (recopi ETOR) / 1 = Fermé*)
	Type_Consigne		:BOOL;	(*Choix du TYPE de pilotage du registre / 1 = ANA / 0 = TOR*)
	Control_Discordance	:BOOL;	(*Autorisation de marche des alarmes / 1 = Alarme autorisé*)
	Tempo_AL_Discor	:TIME;	(*Temporisation pour les alarmes discodance / en sec*)
	Hyst_AL_Discor		:REAL;	(*HystéRésis pour les alarmes discodance si LE registre est en pilotage ANA / en %*)
	Presence_Fdc		:INT;	(*Mot de présence des fin de course / 0 = Pas de fin de course / 1 = Fin de course Ouvert / 2 = Fin de course Fermé / 3 = Les 2 fin de course*)
	Inverse_SAN			:BOOL;	(*Inversion de la sortie SAN / 1 = Sens inverse / 0 = Sens normal*)
	SAN_MIN			:REAL;	(*Valeur minimal de la sortie SAN / en point automate*)
	SAN_MAX			:REAL;	(*Valeur maximal de la sortie SAN / en point automate*)
END_VAR

VAR_OUTPUT
	SAN_CONS_REG			:REAL;	(*Consigne a appliqué au registre ANA (pour SAN) / en %*)
	STOR_CMD_OUV_REG	:BOOL;	(*Commande a appliqué au registre TOR (pour STOR) / 1 = Ouverture*)
END_VAR

VAR
	TON_1			:TON;
	TON_2			:TON;
	TON_3			:TON;
	TON_4			:TON;
	Request			:BOOL;
	CONS_REG_INT	:REAL;
	CMD_REG_INT	:BOOL;
	CONS_REG		:REAL;
	Adr1			:DINT;
	Adr2			:DINT;
	Adr3			:DINT;
	Adr4			:DINT;
	Adr5			:DINT;
	Adr6			:DINT;
	Adr7			:DINT;
	val_x			:REAL;
	val_b			:REAL;
	val_a			:REAL;
	val_y			:REAL;
	val_final			:REAL;
END_VAR

VAR_IN_OUT
	Tab_RegMoto	:Objet_Registre; (*Tableau des valeurs*)
END_VAR

(* Gestion consigne **************************************************************)
IF Tab_RegMoto.Mot_Lecture.5 (* Gestion consigne pour un registre ANA *)
	THEN
		STOR_CMD_OUV_REG := FALSE;
		IF Tab_RegMoto.Mot_Ecriture.0
			THEN
				CONS_REG_INT := Tab_RegMoto.W_ConsForcage;
			ELSE
				CONS_REG_INT := LIMIT(Tab_RegMoto.W_LimiteMinPosition,Cons_Pos_Dem,Tab_RegMoto.W_LimiteMaxPosition);
		END_IF;
		CONS_REG := CONS_REG_INT;
	ELSE (* Gestion consigne pour un registre TOR *)
		CONS_REG := 0.0;
		IF Tab_RegMoto.Mot_Ecriture.0
			THEN
				CMD_REG_INT := Tab_RegMoto.Mot_Ecriture.1;
			ELSE
				CMD_REG_INT := Cmd_Ouv_Dem;
		END_IF;
		STOR_CMD_OUV_REG := CMD_REG_INT;
END_IF;


(* Gestion sortie analogique **************************************************************)
(* Mise à l'echelle sortie ****)
val_x := CONS_REG;
val_b := SAN_Max - (val_a * 100.0);
val_a := (SAN_Max - SAN_Min) / 100.0;
val_y := (val_a * val_x) + val_b;

(* Inversion de la sortie ANA ****)
IF (Inverse_SAN)
	THEN
		val_final := SAN_Max - val_y;
	ELSE
		val_final := val_y;
END_IF;
SAN_CONS_REG := LIMIT(SAN_Min,val_final, SAN_Max);


(* Gestion alarme **************************************************************)
IF Control_Discordance
	THEN
		IF NOT(Type_Consigne) (* Alarme discordance pour registre STOR *)
			THEN
				CASE Presence_Fdc OF
					0 :
						Tab_RegMoto.Mot_Lecture.4 := FALSE;
					1 :
						TON_1(IN := Tab_RegMoto.Mot_Lecture.0 AND NOT(Tab_RegMoto.Mot_Lecture.1),PT := Tempo_AL_Discor);
						Tab_RegMoto.Mot_Lecture.4 := TON_1.Q;

					2 :
						TON_2(IN := NOT(Tab_RegMoto.Mot_Lecture.0) AND NOT(Tab_RegMoto.Mot_Lecture.2),PT := Tempo_AL_Discor);
						Tab_RegMoto.Mot_Lecture.4 := TON_2.Q;

					3 :
						TON_3(IN := (Tab_RegMoto.Mot_Lecture.0 AND NOT(Tab_RegMoto.Mot_Lecture.1)) OR (NOT(Tab_RegMoto.Mot_Lecture.0) AND NOT(Tab_RegMoto.Mot_Lecture.2)),PT := Tempo_AL_Discor);
						Tab_RegMoto.Mot_Lecture.4 := TON_3.Q;

					ELSE Tab_RegMoto.Mot_Lecture.4 := FALSE;

				END_CASE;

			ELSE (* Alarme discordance pour registre SAN *)
				TON_4(IN := ((Tab_RegMoto.R_Position + Hyst_AL_Discor) < Tab_RegMoto.R_InfoConsPosition) OR ((Tab_RegMoto.R_Position - Hyst_AL_Discor) > Tab_RegMoto.R_InfoConsPosition),PT := Tempo_AL_Discor);
				Tab_RegMoto.Mot_Lecture.4 := TON_4.Q;
		END_IF;
ELSE (* Si control discordance désactivé *)
Tab_RegMoto.Mot_Lecture.4 := FALSE;
END_IF;

(* Recopie pour lecture GTC *********************************************************)
Tab_RegMoto.Mot_Lecture.0		:= STOR_CMD_OUV_REG;
Tab_RegMoto.Mot_Lecture.1		:= Info_Fdc_ouvert;
Tab_RegMoto.Mot_Lecture.2		:= Info_Fdc_ferme;
Tab_RegMoto.Mot_Lecture.3 		:= Control_Discordance;
Tab_RegMoto.Mot_Lecture.5		:= Type_Consigne;
Tab_RegMoto.R_Position			:= Info_Mess_Pos;
Tab_RegMoto.R_InfoConsPosition	:= CONS_REG;

END_FUNCTION_BLOCK

// ---- POUs/Block/Autres/Blinck_V2.TcPOU
FUNCTION_BLOCK Blinck_V2
VAR_INPUT
	Enable: BOOL;
	In_Pause: BOOL;
	Timer_Seconde_ON: REAL;
	Timer_Minute_ON: REAL;
	Timer_Heure_ON: REAL;
	Timer_Jour_ON: REAL;
	Timer_Seconde_OFF: REAL;
	Timer_Minute_OFF: REAL;
	Timer_Heure_OFF: REAL;
	Timer_Jour_OFF: REAL;
	Contact_Off: BOOL;
	Contact_On: BOOL;
END_VAR
VAR_OUTPUT
	Out: BOOL;
END_VAR
VAR
	TON_1: TON_V1;
	TON_2: TON_V1;
	Out2: BOOL;
	Out3: BOOL;
END_VAR

TON_1(
    Enable := Enable AND Out2 AND Out3 AND Contact_Off,
    Pause := In_Pause,
    In_Cons_Seconde := Timer_Seconde_OFF,
    In_Cons_Minute := Timer_Minute_OFF,
    In_Cons_Heure := Timer_Heure_OFF,
    In_Cons_Jour := Timer_Jour_OFF); // TON_V1
Out2 := NOT TON_1.Q;
TON_2(
    Enable := Out2 AND Enable AND Contact_On,
    Pause := In_Pause,
    In_Cons_Seconde := Timer_Seconde_ON,
    In_Cons_Minute := Timer_Minute_ON,
    In_Cons_Heure := Timer_Heure_ON,
    In_Cons_Jour := Timer_Jour_ON); // TON_V1
Out3 := TON_2.Q;
Out := NOT Out3 AND Enable;

END_FUNCTION_BLOCK

// ---- POUs/Block/Autres/PWM.TcPOU
FUNCTION_BLOCK PWM
VAR_INPUT
	ENABLE					:BOOL;		(*Autorisation de marche du bloc / 1 = Marche*)
	IN_BaseTemps			:REAL;		(*Base de temps du PWM / En sec*)
	IN_T_ON_Max			:REAL;		(*Temps à ON max autorisé pour la sortie / En sec*)
	TIME_Temp_ON_Min		:TIME;		(*Temps à ON min autorisé pour la sortie / En TIME*)
	IN_Cons					:REAL;		(*Consigne demandé / 0...100,0 %*)
END_VAR
VAR_OUTPUT
	OUT_PWM				:BOOL;		(*Sortie du PWM / 1 = Marche*)
	OUT_Info_Temps_Cycle	:INT;		(*Temps de cycle restant / En minutes*)
END_VAR
VAR
	Temp_ON				:REAL;
	TP_1					:TP;
	TIME_BaseTemps		:TIME;
	TIME_Temp_ON			:TIME;
	DINT_BaseTemps		:DINT;
	DINT_Temp_ON			:DINT;
	Clignotant_V2_1			:BLINK;
	front						:BOOL;
	Temp_T_ON_voulu		:REAL;
	Temp_ON_bis			:REAL;
END_VAR

IF(ENABLE)
	THEN
		IF (IN_Cons = 0.0)
			THEN
				OUT_PWM := FALSE;
			ELSE
				(* Cacule temps PWM *)
				Temp_T_ON_voulu := IN_T_ON_Max;
				Temp_ON := (IN_BaseTemps / 100.0) * IN_Cons;

				(* Sécurité Temp On Max *)
				IF Temp_ON > Temp_T_ON_voulu
					THEN
						Temp_ON_bis := Temp_T_ON_voulu;
					ELSE
						Temp_ON_bis := Temp_ON;
				END_IF;	

				DINT_BaseTemps := REAL_TO_DINT(IN_BaseTemps);
				TIME_BaseTemps := DINT_TO_TIME(DINT_BaseTemps * DINT#1000);

				DINT_Temp_ON := REAL_TO_DINT(Temp_ON_bis * 10.0);
				TIME_Temp_ON := DINT_TO_TIME(DINT_Temp_ON * DINT#100);

				(* Sécurité si Temp ON < 0.2 sec on n'active pas la sortie *)
				IF TIME_Temp_ON > TIME_Temp_ON_Min
					THEN
						Clignotant_V2_1(ENABLE:= TRUE, TIMELOW:=T#1s, TIMEHIGH:=TIME_BaseTemps);
						front := Clignotant_V2_1.OUT;

						TP_1(IN := front,PT := TIME_Temp_ON);
						OUT_PWM := TP_1.Q;
					ELSE
						OUT_PWM := FALSE;
				END_IF;

		END_IF;
	ELSE
		OUT_PWM := FALSE;
END_IF;

END_FUNCTION_BLOCK

// ---- POUs/Block/Cabines/Gache.TcPOU
FUNCTION_BLOCK Gache
VAR_INPUT
	Cmd_Gache 	:BOOL; (*Commande de la prise*)
	Reset_Gache	:BOOL; (*Commande reset du défaut de discordance*)
	Enable_Forcage :BOOL;
	Forcage :BOOL;
END_VAR
VAR_OUTPUT
	STOR_Gache	:BOOL; (*Commande de la sortie TOR de la Gache*)
	Def_Discord_Gache	:BOOL; (*Statut défaut discordance Gache*)
END_VAR
VAR
	TON_1: 				TON;
	RS_1: 				RS;
END_VAR

(*============================Gestion de la commande de la gache================================*)
IF (Enable_Forcage)
	THEN
	IF(Forcage  AND NOT Def_Discord_Gache)
		THEN
		STOR_Gache := TRUE;
		ELSE
		STOR_Gache := FALSE;
	END_IF;
	ELSE
	IF (Cmd_Gache  AND NOT Def_Discord_Gache)
		THEN
		STOR_Gache := TRUE;
		ELSE
		STOR_Gache := FALSE;
	END_IF;
END_IF;

(*============================Gestion défaut discordance gache================================*)
TON_1(IN:= ( FALSE(*STOR_Gache AND NOT Statut_Porte*))  , PT:= t#5s );
RS_1(SET:= TON_1.Q, RESET1:= Reset_Gache);
Def_Discord_Gache := RS_1.Q1;

END_FUNCTION_BLOCK

// ---- POUs/Block/Objets/Objet_Mot_TOR_V1.TcPOU
FUNCTION_BLOCK Objet_Mot_TOR_V1
VAR_INPUT
	Cmd_Ma_Moteur			:BOOL;	(*Commande de la marche du moteur / 1 = Marche*)
	Info_ETOR_Ma_Moteur	:BOOL;	(*Information TOR de la marche du moteur / 1 = Marche*)
	Info_ETOR_Def_Moteur	:BOOL;	(*Information TOR du défaut du moteur / 1 = Défaut*)
END_VAR

VAR_OUTPUT
	STOR_CMD_MOTEUR	:BOOL;	(*Commande ouverture a appliqué au Moteur (pour STOR) / 1 = Marche*)
END_VAR

VAR_IN_OUT
	Tab_MoteurTOR	:Objet_Mot_TOR; (*Tableau des valeurs*)
END_VAR

(* Recopie pour lecture GTC *********************************************************)
Tab_MoteurTOR.Mot_Lecture.0		:= STOR_CMD_MOTEUR;
Tab_MoteurTOR.Mot_Lecture.2   	:= Info_ETOR_Ma_Moteur;
Tab_MoteurTOR.Mot_Lecture.1  		:= Info_ETOR_Def_Moteur;

(* Gestion commande **************************************************************)
IF Tab_MoteurTOR.Mot_Ecriture.0
	THEN
		STOR_CMD_MOTEUR := Tab_MoteurTOR.Mot_Ecriture.1;
	ELSE
		STOR_CMD_MOTEUR := Cmd_Ma_Moteur;
END_IF;

END_FUNCTION_BLOCK

// ---- POUs/Block/Objets/Objet_PI_V1.TcPOU
FUNCTION_BLOCK Objet_PI_V1
VAR_INPUT
	Cons_Variable			:REAL;	(*Consigne variable Régulante / L'unité dépend de la régulation (°C / % / Pa / bar / m3/h / mg/l ect ....)*)
	Mes_Regul				:REAL;	(*Mesure Régulante / L'unité dépend de la régulation (°C / % / Pa / bar / m3/h / mg/l ect ....)*)
	Autorisation_Marche		:BOOL;	(*Autorisation marche Régulation / 1 = Marche*)
	Type_Consigne			:BOOL;	(*TYPE consigne Régulation /  0 = Variable / 1 = Fixe (Fonctionne avec Consigne Occupé/Inoccupé)*)
	SelConsigneInoccupe		:BOOL;	(*1 = Fonctionnement uniquement sur consigne Inoccupé / 0 = Consigne occupé / inoccupé*)
	Mode_Occupe			:BOOL;	(*Mode occupé/inoccupé / 1 = Occupé / 0 = Inoccupé*)
	Sens_PID				:BOOL;	(*Sens du PID / 1 = FROID / 0 = CHAUD*)
	MIN_Sortie_CMD_PID		:REAL;	(*Limite MIN Sortie commande Régulation / L'unité dépend de la régulation (°C / % / Pa / bar / m3/h / mg/l ect ....)*)
	MAX_Sortie_CMD_PID		:REAL;	(*Limite MAX Sortie commande Régulation / L'unité dépend de la régulation (°C / % / Pa / bar / m3/h / mg/l ect ....)*)
	Gain_Variable			:BOOL;	(*Activation du gain variable / 1 = Gain variable activé*)
	Hyst_Gain_Variable		:REAL;	(*HystéRésis d'enclenchement du Gain variable / L'unité dépend de la Régulation (°C / % / Pa / bar / m3/h / mg/l ect ....)*)
	Coef_Gain_Variable		:REAL;	(*Coéficient multiplicateur du Gain variable / En %*)
	EN_Filtre_S_CMD_PID		:BOOL;	(*Activation du filtre de la sortie commande PID / 1 = Filtre actif*)
	Tempo_Puls_Filtre		:TIME;	(*Temporisation entre chaque pulse pour LE filtrage de la sortie commande / En sec*)
	IN_UP_RATE				:REAL;	(*Echellon d'incrementation de la sortie commande PID / 0...100,0 %*)
	IN_DOWN_RATE			:REAL;	(*Echellon décrémentation de la sortie commande PID / 0...100,0 %*)
	EN_Mes_pertub			:BOOL;	(*Activation de la compensation de mesure de perturbation / 1 = Activé*)
	Coef_Mes_pertub			:REAL;	(*Coéficient multiplicateur de la mesure de perturbation / En %*)
	Mesure_pertub			:REAL;	(*Mesure de perturbation*)
	Temps_Perturbation		:TIME;	(*Temporisation d'échantillonage pour la mesure perturbation / En sec*)
END_VAR

VAR_OUTPUT
	Sortie_CMD_PID			:REAL;	(*Sortie commande Régulation / L'unité dépend de la régulation (°C / % / Pa / bar / m3/h / mg/l ect ....)*)
	Sortie_CMD_PID_Brute		:REAL;	(*Sortie commande Régulation apréS bloc PID / L'unité dépend de la régulation (°C / % / Pa / bar / m3/h / mg/l ect ....)*)
	Gain					:REAL;	(*Info du gain Séléctionné pour LE PID*)
	Ecart_Mesure_Cons		:REAL;	(*Info de l'écart de consigne entre la mesure et la consigne*)
END_VAR

VAR
	TON_Filtre			:TON;
	TP_Filtre				:TP;
	TON_Pertub			:TON;
	TP_Pertub			:TP;
	R_TRIG_Pertub		:R_TRIG;
	R_TRIG_1			:R_TRIG;
	Cons_PID_INT		:REAL;
	Cons_PID_INT2		:REAL;
	Status_Marche		:BOOL;
	CONS_Filtrer			:REAL; (*Sortie lissé / 0...100,0 %*)
	CONS_OLD			:REAL; (*0...100,0 % / 0...100,0*)
	PULS_Filtre			:BOOL;
	Gain_Mes_pertub		:REAL; (*Gain calculé pour la mesure de perturbation*)
	Gain_Int				:REAL; (*Info du gain séléctionné pour le PID*)
	Mesure_pertub_old	:REAL;
	Diff_Mesure_pertub	:REAL;
	puls_detecte			:BOOL;
	FPID_1				: PID;
	Calcul1				:REAL;
END_VAR

VAR_IN_OUT
	Tab_RegulPI	:Objet_RegulPI; (*Tableau des valeurs*)
END_VAR

(* Gestion autorisation marche *********************************************************)
Status_Marche := Autorisation_Marche;

(* Gestion consigne régulante *********************************************************)
(* Selection consigne *)
IF Tab_RegulPI.Mot_Lecture.3
	THEN
		Cons_PID_INT := Tab_RegulPI.W_ConsInoccupe;
	ELSE
		IF NOT(Tab_RegulPI.Mot_Lecture.1)
			THEN
				Cons_PID_INT := Cons_Variable;
			ELSE
				IF Tab_RegulPI.Mot_Lecture.2
					THEN
						Cons_PID_INT := Tab_RegulPI.W_ConsOccupe;
					ELSE
						Cons_PID_INT := Tab_RegulPI.W_ConsInoccupe;
				END_IF;
		END_IF;
END_IF;

(* Intégration de la bande morte *)
IF Sens_PID
	THEN
		Cons_PID_INT2 := Cons_PID_INT + Tab_RegulPI.W_BandeMorte;
	ELSE
		Cons_PID_INT2 := Cons_PID_INT - Tab_RegulPI.W_BandeMorte;
END_IF;

(* Forçage consigne *)
IF Tab_RegulPI.Mot_Ecriture.0
	THEN
		Tab_RegulPI.R_InfoConsPI := Tab_RegulPI.W_ConsPIForcage;
	ELSE
		Tab_RegulPI.R_InfoConsPI := LIMIT(Tab_RegulPI.W_LimiteMinCons,Cons_PID_INT2,Tab_RegulPI.W_LimiteMaxCons);
END_IF;

(*  Gestion mesure perturbation *)
R_TRIG_Pertub(CLK := TP_Pertub.Q);
IF R_TRIG_Pertub.Q
	THEN
		Diff_Mesure_pertub := ABS(Mesure_pertub - Mesure_pertub_old);
		Mesure_pertub_old := Mesure_pertub;
END_IF;
IF ((Coef_Mes_pertub * Diff_Mesure_pertub) = 0.0)
	THEN 
		Gain_Mes_pertub := 1.0;
	ELSE
		Gain_Mes_pertub := Coef_Mes_pertub * Diff_Mesure_pertub;	
END_IF;

(* Séléction du gain PID *)
IF Gain_Variable
	THEN
		IF ((Tab_RegulPI.R_MesRegulPI >= (Tab_RegulPI.R_InfoConsPI - Hyst_Gain_Variable)) AND (Tab_RegulPI.R_MesRegulPI <= (Tab_RegulPI.R_InfoConsPI + Hyst_Gain_Variable)))
			THEN
				Gain_Int := Tab_RegulPI.W_GainPI * Coef_Gain_Variable;
			ELSE
				Gain_Int := Tab_RegulPI.W_GainPI;
		END_IF;
	ELSE
		Gain_Int := Tab_RegulPI.W_GainPI;	
END_IF;

IF EN_Mes_pertub
	THEN
		Gain := Gain_Int / Gain_Mes_pertub;
	ELSE
		Gain := Gain_Int;
END_IF;

(* Sens du PID(Inversion du signe du gain) *********************************************************)
IF (Sens_PID)
	THEN
	Gain := 0.0 - Gain;
	ELSE
	Gain := Gain;
END_IF

(* Régulation PID *********************************************************)
FPID_1(
	ACTUAL:= 		Tab_RegulPI.R_MesRegulPI,
	SET_POINT:= 	Tab_RegulPI.R_InfoConsPI,
	KP:= 			Gain,
	TN:= 			Tab_RegulPI.W_IntegralPI,
	TV:= 			Tab_RegulPI.W_DerivPI,
	Y_MANUAL:= 	0.0,
	Y_OFFSET:= 		0.0,
	Y_MIN:= 			MIN_Sortie_CMD_PID,
	Y_MAX:= 		MAX_Sortie_CMD_PID,
	RESET:= 		NOT Status_Marche);
Ecart_Mesure_Cons := FPID_1.ERROR;

(* Gestion sortie commande PID *********************************************************)
IF Tab_RegulPI.Mot_Ecriture.1
	THEN
		Tab_RegulPI.R_SortieCmdPI := Tab_RegulPI.W_SortieCMDForcage;
	ELSE
		IF Tab_RegulPI.Mot_Lecture.0
			THEN
				IF NOT(EN_Filtre_S_CMD_PID)
					THEN
						Tab_RegulPI.R_SortieCmdPI := FPID_1.Y;
					ELSE (* Filtrage sortie commande PID *)
					(* Detection de front montant *)
					R_TRIG_1(CLK := PULS_Filtre);
					puls_detecte := R_TRIG_1.Q;
 
					IF (puls_detecte)
						THEN
							IF (FPID_1.Y > CONS_OLD)
								THEN
									CONS_Filtrer := CONS_Filtrer + IN_UP_RATE;
									CONS_OLD := CONS_Filtrer;
							END_IF;
							IF (FPID_1.Y < CONS_OLD)
								THEN
									CONS_Filtrer := CONS_Filtrer - IN_DOWN_RATE;
									CONS_OLD := CONS_Filtrer;
							END_IF;
							IF (FPID_1.Y = 100.0)
								THEN
									CONS_Filtrer := CONS_Filtrer + IN_UP_RATE;
									CONS_OLD := CONS_Filtrer;
							END_IF;
							IF (FPID_1.Y = 0.0)
								THEN
									CONS_Filtrer := CONS_Filtrer - IN_DOWN_RATE;
									CONS_OLD := CONS_Filtrer;
							END_IF;
					END_IF;
					Tab_RegulPI.R_SortieCmdPI := LIMIT(MIN_Sortie_CMD_PID,CONS_Filtrer,MAX_Sortie_CMD_PID);
				END_IF;
			ELSE
				Tab_RegulPI.R_SortieCmdPI := 0.0;
		END_IF;
END_IF;
Sortie_CMD_PID := Tab_RegulPI.R_SortieCmdPI;
Sortie_CMD_PID_Brute := FPID_1.Y;

(* Recopie pour lecture GTC *********************************************************)
Tab_RegulPI.R_MesRegulPI	:= Mes_Regul;
Tab_RegulPI.Mot_Lecture.0	:= Status_Marche;
Tab_RegulPI.Mot_Lecture.1 	:= Type_Consigne;
Tab_RegulPI.Mot_Lecture.2	:= Mode_Occupe;
Tab_RegulPI.Mot_Lecture.3 	:= SelConsigneInoccupe;

END_FUNCTION_BLOCK

// ---- POUs/Block/Objets/Objet_Pressostat_V1.TcPOU
FUNCTION_BLOCK Objet_Pressostat_V1
VAR_INPUT
	Info_Pressostat	:BOOL;	(*nfo détection préssostat / 1 = Détection*)
	Seuil_Press		:REAL;	(*Seuil préssion Réglé sur LE préssostat / en Pa*)
END_VAR
VAR_OUTPUT
END_VAR
VAR
	R_StatDefaut: BOOL;
	R_SeuilPress: REAL;
END_VAR
VAR_IN_OUT
	Tab_Pressostat: Objet_Pressostat;
END_VAR

(* Gestion mesure **************************************************************)
R_StatDefaut	:= Info_Pressostat;
Tab_Pressostat.R_SeuilPress	:= Seuil_Press;

(* Gestion lecture GTC *********************************************************)
Tab_Pressostat.Mot_Lecture.0:= R_StatDefaut;

END_FUNCTION_BLOCK

// ---- Visualizations/Visualizations/GestionAlarme/Programme/GestionAlarme.TcPOU
PROGRAM GestionAlarme
VAR CONSTANT
	nbErreurMax 					: INT := 500; //définit le nombre d'erreur maximum que l'on peur gérer	
	IndexDepartWarning  			: INT := 250;  //Définit l'index de départ des warning dans la liste d'erreur
	IndexDepartWarningAcquittable  	: INT := 375;  //Définit l'index de départ des warning toujours aquittable dans la liste d'erreur
	nbErreurMaxHistorique 			: INT := 1000; //définit le nombre d'erreur maximum que l'on peut inscrire dans l'historique	
END_VAR
VAR
	TableauErreurRaw 	: ARRAY[0..nbErreurMax] OF Erreur_Struct; //Contiendra les erreurs dans l'ordre d'arrivé
	TableauErreurVisu	: ARRAY[0..nbErreurMax] OF Erreur_StructVisu; //Contiendra les erreurs formatées
	TextlistErreur 		: ARRAY[0..nbErreurMax] OF BOOL;
	TextlistErreurOLD 	: ARRAY[0..nbErreurMax] OF BOOL;
	index: INT;
	NbrErreur: INT;
	NT_GetTime1: NT_GetTime;
	DateEnCour: DATE_AND_TIME;
	// Bouton pour l'aquittement des défauts
	bAcquitement: BOOL;
	// représente la ligne en cour de sélection dans la visu
	indexLigneActive: INT;
	// bouton d'aquittement de tout les défauts
	bAcquitementAll: BOOL;
	index3: INT;
	index4: INT;
	index2: INT;
	NbrErreurSave: INT;
	DateEncourString: STRING;
	tickDate: BOOL;
	// Permet l'affichage croissant ou decroissant des défauts
	bOrdreCroissant: BOOL;
	LigneSelectionTabVisu: INT;
	DernierDefautIDVisu: INT;
	DernierDefautIDImageVisu: STRING(3);
	CouleurBandeauVisu: DWORD;
	bAckBandeau: BOOL;
	// sera liée à la visu pour éviter les indexs négatifs
	NbrErreurVisu: INT;
	// sera liée à la visu pour éviter les indexs négatifs
	nombredefautHistoriqueVisu: INT;
	sDay:	STRING;
	sMonth:	STRING;
	sYear:	STRING;
	sHour:	STRING;
	sMinute:STRING;
	sSecond:STRING;
END_VAR

VAR PERSISTENT
	HistoriqueDefaut : ARRAY[0..nbErreurMaxHistorique] OF Erreur_StructVisu;
	nombredefautHistorique : INT;
END_VAR

(*///////////////////////////////////////////////////////////////////////////////////////////////////////////////////////////////////////////////////////////////////////////////////
Programme d'exemple d'utilisation des alarmes
Date : 25-09-2015
Auteur : Jerome CHOVINO
Version : V1.1

Résumé : 	On peut gérer trois catégories (erreurs, warning et warning acquittables), il faut modifier la textlist "listeErreurWarning" pour créer les textes d'erreur
			et mettre le bon booléen dans le tableau d'erreur définit dans l'action "DefinitionIDErreur" en face de l'index case tableau qui correspond à l'index de la textlist.
			/!\ L'index 0 de la textlist "listeErreurWarning" doit rester vide !
			
/////////////////////////////////////////////////////////////////////////////////////////////////////////////////////////////////////////////////////////////////////////////////////*)

DefinitionIDErreur(); //Actualisation des défauts
//Recupération de la date en cour (utilise la librairie TC2_Utilities)
tickDate := NOT tickDate;
NT_GetTime1(
	START:= tickDate, 
	TMOUT:= T#200MS);
//Contruction de la date en string
sDay:=WORD_TO_STRING(NT_GetTime1.TIMESTR.wDay);
IF len(sDAy)< 2 THEN sday:= concat('0',sday) ; END_IF

sMonth:=WORD_TO_STRING(NT_GetTime1.TIMESTR.wMonth);
IF len(sMonth)< 2 THEN sMonth:= concat('0',sMonth) ; END_IF

sYear:=WORD_TO_STRING(NT_GetTime1.TIMESTR.wYear);
IF len(sYear)< 2 THEN sYear:= concat('0',sYear) ; END_IF

sHour:=WORD_TO_STRING(NT_GetTime1.TIMESTR.wHour);
IF len(sHour)< 2 THEN sHour:= concat('0',sHour) ; END_IF

sMinute:=WORD_TO_STRING(NT_GetTime1.TIMESTR.wMinute);
IF len(sMinute)< 2 THEN sMinute:= concat('0',sMinute) ; END_IF

sSecond:=WORD_TO_STRING(NT_GetTime1.TIMESTR.wSecond);
IF len(sSecond)< 2 THEN sSecond:= concat('0',sSecond) ; END_IF

DateEncourString := sday;
DateEncourString := CONCAT(DateEncourString,'/');
DateEncourString := CONCAT(DateEncourString,sMonth);
DateEncourString := CONCAT(DateEncourString,'/');
DateEncourString := CONCAT(DateEncourString,sYear);
DateEncourString := CONCAT(DateEncourString,'  ');
DateEncourString := CONCAT(DateEncourString,sHour);
DateEncourString := CONCAT(DateEncourString,':');
DateEncourString := CONCAT(DateEncourString,sMinute);
DateEncourString := CONCAT(DateEncourString,':');
DateEncourString := CONCAT(DateEncourString,sSecond);

//Structation des erreurs
FOR index := 0 TO nbErreurMax DO 
	//Nouveau défaut
	IF TextlistErreur[index] AND NOT TextlistErreurOLD[index]  THEN		
		TableauErreurRaw[NbrErreur].IdDefaut := index;		
		TableauErreurRaw[NbrErreur].DateDefaut := 	DateEncourString;
		IF index >= IndexDepartWarningAcquittable THEN //Warnings Acquittables
			TableauErreurRaw[NbrErreur].TypeDefaut := 2; //1 = Warning acquittable, voir structure Erreur_Struct
			TableauErreurRaw[NbrErreur].EtatDefaut := 'WA'; //nouveau warning acquittable 
		ELSIF index >= IndexDepartWarning THEN //Warnings
			TableauErreurRaw[NbrErreur].TypeDefaut := 1; //1 = Warning, voir structure Erreur_Struct
			TableauErreurRaw[NbrErreur].EtatDefaut := 'WP'; //nouveau warning 
		ELSE //Erreurs
			TableauErreurRaw[NbrErreur].TypeDefaut := 0; //0 = Erreur, voir structure Erreur_Struct
			TableauErreurRaw[NbrErreur].EtatDefaut := 'DP'; //nouveau Defaut 
		END_IF
	
		//Ajout du nouveau défaut dans l'historique des défauts
		HistoriqueDefaut[nombredefautHistorique].DateMessage := TableauErreurRaw[NbrErreur].DateDefaut;
		HistoriqueDefaut[nombredefautHistorique].IDMessage := TableauErreurRaw[NbrErreur].IdDefaut;
		HistoriqueDefaut[nombredefautHistorique].TypeDefaut := TableauErreurRaw[NbrErreur].EtatDefaut;
		nombredefautHistorique := nombredefautHistorique + 1;
		IF nombredefautHistorique > nbErreurMaxHistorique THEN nombredefautHistorique := 0; END_IF	
		
		NbrErreur := NbrErreur + 1;
		IF NbrErreur > nbErreurMax THEN NbrErreur := 0; END_IF					
	END_IF	
	
	TextlistErreurOLD[index] := TextlistErreur[index];	
END_FOR

FOR index := NbrErreur TO nbErreurMax DO //Effacer les cases vides du tableau brute
	TableauErreurRaw[index].IdDefaut := 0;	
	TableauErreurRaw[index].EtatDefaut := '';
END_FOR

//MAJ de l'état des défauts
//Défaut disparu non acquité (ne s'applique pas aux warnings acquittables)
FOR index := 0 TO NbrErreur DO
	IF NOT TextlistErreur[TableauErreurRaw[index].IdDefaut] AND (TableauErreurRaw[index].IdDefaut <> 0)  AND (TableauErreurRaw[index].TypeDefaut <> 2) THEN	
		IF TableauErreurRaw[index].IdDefaut < IndexDepartWarning THEN //Erreur
			TableauErreurRaw[index].EtatDefaut := 'DD'; //nouveau Defaut 
		ELSE//Warning
			TableauErreurRaw[index].EtatDefaut := 'WD'; //nouveau warning 
		END_IF		
	END_IF
END_FOR


//Acquittement des défauts sélectionnés
IF bAcquitement THEN
	bAcquitement := FALSE;
	//On ne peut aquitter que les défauts qui ont disparu ou les warning aquittable
	IF (TableauErreurRaw[indexLigneActive].IdDefaut <> 0) AND ( NOT TextlistErreur[TableauErreurRaw[indexLigneActive].IdDefaut] OR (TableauErreurRaw[indexLigneActive].TypeDefaut = 2) ) THEN
		FOR index := indexLigneActive TO NbrErreur DO 
			TableauErreurRaw[index] :=  TableauErreurRaw[index + 1];	
		END_FOR	
		NbrErreur := NbrErreur - 1;
		IF NbrErreur < 0 THEN NbrErreur := 0; END_IF
	END_IF
END_IF


//Acquittement de tous les défauts
IF bAcquitementAll THEN
	bAcquitementAll := FALSE;
	NbrErreurSave := NbrErreur;
	index2 := 0 ;
	FOR index := 0 TO NbrErreurSave DO 
		//On ne peut aquitter que les défauts qui ont disparu ou les warning aquittable
		IF (TableauErreurRaw[index2].IdDefaut <> 0) AND (NOT TextlistErreur[TableauErreurRaw[index2].IdDefaut] OR (TableauErreurRaw[index2].TypeDefaut = 2) ) THEN
			FOR index3 := index2 TO NbrErreur DO 
				TableauErreurRaw[index3] :=  TableauErreurRaw[index3 + 1];	
			END_FOR	
			NbrErreur := NbrErreur - 1;
			IF NbrErreur < 0 THEN NbrErreur := 0; END_IF
		ELSE
			index2 := index2 + 1;
			IF index2 > NbrErreurSave  THEN  index2 := NbrErreurSave; END_IF	
		END_IF
	END_FOR	
END_IF

//Mise en forme pour affichage dans la visu
//Tableau d'alarme
IF NOT bOrdreCroissant THEN
	FOR index:=0 TO NbrErreur DO
		TableauErreurVisu[index].TypeDefaut := TableauErreurRaw[index].EtatDefaut;
		TableauErreurVisu[index].IDMessage := TableauErreurRaw[index].IdDefaut;
		TableauErreurVisu[index].DateMessage := TableauErreurRaw[index].DateDefaut;
	END_FOR
	indexLigneActive := LigneSelectionTabVisu; //Variable liée au tableau de la visu
ELSE
	FOR index:=NbrErreur-1 TO 0 BY -1 DO 
		TableauErreurVisu[index].TypeDefaut := TableauErreurRaw[(NbrErreur-1) - index].EtatDefaut;
		TableauErreurVisu[index].IDMessage := TableauErreurRaw[(NbrErreur-1) - index].IdDefaut;
		TableauErreurVisu[index].DateMessage := TableauErreurRaw[(NbrErreur-1) - index].DateDefaut;
	END_FOR	
	indexLigneActive := (NbrErreur-1)- LigneSelectionTabVisu; //Variable liée au tableau de la visu
END_IF
IF NbrErreur <= 0 THEN NbrErreurVisu := 1; ELSE NbrErreurVisu := NbrErreur; END_IF
	
//Historique d'alarme
//Bandeau d'alarme
IF NbrErreur > 0 THEN
	DernierDefautIDVisu := TableauErreurRaw[NbrErreur-1].IdDefaut;
	DernierDefautIDImageVisu := TableauErreurRaw[NbrErreur-1].EtatDefaut;
	//Le changement de couleur n'est pas fonctionnel avec la version 4018.13
	IF 		TableauErreurRaw[NbrErreur-1].EtatDefaut = 'DP' THEN CouleurBandeauVisu := 16#00FF0000; //Bandeau rouge
	ELSIF 	TableauErreurRaw[NbrErreur-1].EtatDefaut = 'DD' THEN CouleurBandeauVisu := 16#00FF0066; //Bandeau Rouge clair
	ELSIF 	TableauErreurRaw[NbrErreur-1].EtatDefaut = 'WP' THEN CouleurBandeauVisu := 16#00FF6600; //Bandeau orange
	ELSIF 	TableauErreurRaw[NbrErreur-1].EtatDefaut = 'WD' THEN CouleurBandeauVisu := 16#00FF9966; //Bandeau orange clair 
	ELSIF 	TableauErreurRaw[NbrErreur-1].EtatDefaut = 'WA' THEN CouleurBandeauVisu := 16#003366FF; //Bandeau Bleu
	END_IF
ELSE
	DernierDefautIDVisu := 0;
	DernierDefautIDImageVisu := '0';
	CouleurBandeauVisu := 16#00FFFFFF; //Bandeau blanc
END_IF
IF nombredefautHistorique <= 0 THEN nombredefautHistoriqueVisu := 1; ELSE nombredefautHistoriqueVisu := nombredefautHistorique; END_IF

//Bandeau alarme
IF bAckBandeau THEN
	bAckBandeau := FALSE;
	IF NbrErreur>0 THEN
	//On ne peut aquitter que les défauts qui ont disparu ou les warning aquittable
		IF (TableauErreurRaw[NbrErreur-1].IdDefaut <> 0) AND (NOT TextlistErreur[TableauErreurRaw[NbrErreur-1].IdDefaut] OR (TableauErreurRaw[NbrErreur-1].TypeDefaut = 2)) THEN
			TableauErreurRaw[NbrErreur-1] :=  TableauErreurRaw[index + 1];	
			NbrErreur := NbrErreur - 1;
			IF NbrErreur < 0 THEN NbrErreur := 0; END_IF
		END_IF	
	END_IF	
END_IF

ACTION DefinitionIDErreur:
//Fait le lien entre la text list et la variable PLC booléenne qui remonte l'erreur ou les warning
//Les erreurs vont de l'index 1 à 249  -> Acquittable que si le défaut n'est plus la
//Les warnings de 250 à 374 -> Acquittable que si le warning n'est plus la, voir constante "IndexDepartWarning"
//Les warnings Acquittables de 375 à 499 -> Acquittable dans tout les cas "IndexDepartWarningAcquittable"


//Erreurs 
TextlistErreur[	1	]	 := ErreurPuissance;
TextlistErreur[	2	]	 := ErreurAXE1;
TextlistErreur[	3	]	 := ErreurAXE2;
TextlistErreur[	4	]	 := ErreurXTS;
TextlistErreur[	5	]	 := ErreurAir;
(*
TextlistErreur[	6	]	 := ;
TextlistErreur[	7	]	 := ;
TextlistErreur[	8	]	 := ;
TextlistErreur[	9	]	 := ;
TextlistErreur[	10	]	 := ;
TextlistErreur[	11	]	 := ;
TextlistErreur[	12	]	 := ;
TextlistErreur[	13	]	 := ;
TextlistErreur[	14	]	 := ;
TextlistErreur[	15	]	 := ;
TextlistErreur[	16	]	 := ;
TextlistErreur[	17	]	 := ;
TextlistErreur[	18	]	 := ;
TextlistErreur[	19	]	 := ;
TextlistErreur[	20	]	 := ;
TextlistErreur[	21	]	 := ;
TextlistErreur[	22	]	 := ;
TextlistErreur[	23	]	 := ;
TextlistErreur[	24	]	 := ;
TextlistErreur[	25	]	 := ;
TextlistErreur[	26	]	 := ;
TextlistErreur[	27	]	 := ;
TextlistErreur[	28	]	 := ;
TextlistErreur[	29	]	 := ;
TextlistErreur[	30	]	 := ;
TextlistErreur[	31	]	 := ;
TextlistErreur[	32	]	 := ;
TextlistErreur[	33	]	 := ;
TextlistErreur[	34	]	 := ;
TextlistErreur[	35	]	 := ;
TextlistErreur[	36	]	 := ;
TextlistErreur[	37	]	 := ;
TextlistErreur[	38	]	 := ;
TextlistErreur[	39	]	 := ;
TextlistErreur[	40	]	 := ;
TextlistErreur[	41	]	 := ;
TextlistErreur[	42	]	 := ;
TextlistErreur[	43	]	 := ;
TextlistErreur[	44	]	 := ;
TextlistErreur[	45	]	 := ;
TextlistErreur[	46	]	 := ;
TextlistErreur[	47	]	 := ;
TextlistErreur[	48	]	 := ;
TextlistErreur[	49	]	 := ;
TextlistErreur[	50	]	 := ;
TextlistErreur[	51	]	 := ;
TextlistErreur[	52	]	 := ;
TextlistErreur[	53	]	 := ;
TextlistErreur[	54	]	 := ;
TextlistErreur[	55	]	 := ;
TextlistErreur[	56	]	 := ;
TextlistErreur[	57	]	 := ;
TextlistErreur[	58	]	 := ;
TextlistErreur[	59	]	 := ;
TextlistErreur[	60	]	 := ;
TextlistErreur[	61	]	 := ;
TextlistErreur[	62	]	 := ;
TextlistErreur[	63	]	 := ;
TextlistErreur[	64	]	 := ;
TextlistErreur[	65	]	 := ;
TextlistErreur[	66	]	 := ;
TextlistErreur[	67	]	 := ;
TextlistErreur[	68	]	 := ;
TextlistErreur[	69	]	 := ;
TextlistErreur[	70	]	 := ;
TextlistErreur[	71	]	 := ;
TextlistErreur[	72	]	 := ;
TextlistErreur[	73	]	 := ;
TextlistErreur[	74	]	 := ;
TextlistErreur[	75	]	 := ;
TextlistErreur[	76	]	 := ;
TextlistErreur[	77	]	 := ;
TextlistErreur[	78	]	 := ;
TextlistErreur[	79	]	 := ;
TextlistErreur[	80	]	 := ;
TextlistErreur[	81	]	 := ;
TextlistErreur[	82	]	 := ;
TextlistErreur[	83	]	 := ;
TextlistErreur[	84	]	 := ;
TextlistErreur[	85	]	 := ;
TextlistErreur[	86	]	 := ;
TextlistErreur[	87	]	 := ;
TextlistErreur[	88	]	 := ;
TextlistErreur[	89	]	 := ;
TextlistErreur[	90	]	 := ;
TextlistErreur[	91	]	 := ;
TextlistErreur[	92	]	 := ;
TextlistErreur[	93	]	 := ;
TextlistErreur[	94	]	 := ;
TextlistErreur[	95	]	 := ;
TextlistErreur[	96	]	 := ;
TextlistErreur[	97	]	 := ;
TextlistErreur[	98	]	 := ;
TextlistErreur[	99	]	 := ;
TextlistErreur[	100	]	 := ;
TextlistErreur[	101	]	 := ;
TextlistErreur[	102	]	 := ;
TextlistErreur[	103	]	 := ;
TextlistErreur[	104	]	 := ;
TextlistErreur[	105	]	 := ;
TextlistErreur[	106	]	 := ;
TextlistErreur[	107	]	 := ;
TextlistErreur[	108	]	 := ;
TextlistErreur[	109	]	 := ;
TextlistErreur[	110	]	 := ;
TextlistErreur[	111	]	 := ;
TextlistErreur[	112	]	 := ;
TextlistErreur[	113	]	 := ;
TextlistErreur[	114	]	 := ;
TextlistErreur[	115	]	 := ;
TextlistErreur[	116	]	 := ;
TextlistErreur[	117	]	 := ;
TextlistErreur[	118	]	 := ;
TextlistErreur[	119	]	 := ;
TextlistErreur[	120	]	 := ;
TextlistErreur[	121	]	 := ;
TextlistErreur[	122	]	 := ;
TextlistErreur[	123	]	 := ;
TextlistErreur[	124	]	 := ;
TextlistErreur[	125	]	 := ;
TextlistErreur[	126	]	 := ;
TextlistErreur[	127	]	 := ;
TextlistErreur[	128	]	 := ;
TextlistErreur[	129	]	 := ;
TextlistErreur[	130	]	 := ;
TextlistErreur[	131	]	 := ;
TextlistErreur[	132	]	 := ;
TextlistErreur[	133	]	 := ;
TextlistErreur[	134	]	 := ;
TextlistErreur[	135	]	 := ;
TextlistErreur[	136	]	 := ;
TextlistErreur[	137	]	 := ;
TextlistErreur[	138	]	 := ;
TextlistErreur[	139	]	 := ;
TextlistErreur[	140	]	 := ;
TextlistErreur[	141	]	 := ;
TextlistErreur[	142	]	 := ;
TextlistErreur[	143	]	 := ;
TextlistErreur[	144	]	 := ;
TextlistErreur[	145	]	 := ;
TextlistErreur[	146	]	 := ;
TextlistErreur[	147	]	 := ;
TextlistErreur[	148	]	 := ;
TextlistErreur[	149	]	 := ;
TextlistErreur[	150	]	 := ;
TextlistErreur[	151	]	 := ;
TextlistErreur[	152	]	 := ;
TextlistErreur[	153	]	 := ;
TextlistErreur[	154	]	 := ;
TextlistErreur[	155	]	 := ;
TextlistErreur[	156	]	 := ;
TextlistErreur[	157	]	 := ;
TextlistErreur[	158	]	 := ;
TextlistErreur[	159	]	 := ;
TextlistErreur[	160	]	 := ;
TextlistErreur[	161	]	 := ;
TextlistErreur[	162	]	 := ;
TextlistErreur[	163	]	 := ;
TextlistErreur[	164	]	 := ;
TextlistErreur[	165	]	 := ;
TextlistErreur[	166	]	 := ;
TextlistErreur[	167	]	 := ;
TextlistErreur[	168	]	 := ;
TextlistErreur[	169	]	 := ;
TextlistErreur[	170	]	 := ;
TextlistErreur[	171	]	 := ;
TextlistErreur[	172	]	 := ;
TextlistErreur[	173	]	 := ;
TextlistErreur[	174	]	 := ;
TextlistErreur[	175	]	 := ;
TextlistErreur[	176	]	 := ;
TextlistErreur[	177	]	 := ;
TextlistErreur[	178	]	 := ;
TextlistErreur[	179	]	 := ;
TextlistErreur[	180	]	 := ;
TextlistErreur[	181	]	 := ;
TextlistErreur[	182	]	 := ;
TextlistErreur[	183	]	 := ;
TextlistErreur[	184	]	 := ;
TextlistErreur[	185	]	 := ;
TextlistErreur[	186	]	 := ;
TextlistErreur[	187	]	 := ;
TextlistErreur[	188	]	 := ;
TextlistErreur[	189	]	 := ;
TextlistErreur[	190	]	 := ;
TextlistErreur[	191	]	 := ;
TextlistErreur[	192	]	 := ;
TextlistErreur[	193	]	 := ;
TextlistErreur[	194	]	 := ;
TextlistErreur[	195	]	 := ;
TextlistErreur[	196	]	 := ;
TextlistErreur[	197	]	 := ;
TextlistErreur[	198	]	 := ;
TextlistErreur[	199	]	 := ;
TextlistErreur[	200	]	 := ;
TextlistErreur[	201	]	 := ;
TextlistErreur[	202	]	 := ;
TextlistErreur[	203	]	 := ;
TextlistErreur[	204	]	 := ;
TextlistErreur[	205	]	 := ;
TextlistErreur[	206	]	 := ;
TextlistErreur[	207	]	 := ;
TextlistErreur[	208	]	 := ;
TextlistErreur[	209	]	 := ;
TextlistErreur[	210	]	 := ;
TextlistErreur[	211	]	 := ;
TextlistErreur[	212	]	 := ;
TextlistErreur[	213	]	 := ;
TextlistErreur[	214	]	 := ;
TextlistErreur[	215	]	 := ;
TextlistErreur[	216	]	 := ;
TextlistErreur[	217	]	 := ;
TextlistErreur[	218	]	 := ;
TextlistErreur[	219	]	 := ;
TextlistErreur[	220	]	 := ;
TextlistErreur[	221	]	 := ;
TextlistErreur[	222	]	 := ;
TextlistErreur[	223	]	 := ;
TextlistErreur[	224	]	 := ;
TextlistErreur[	225	]	 := ;
TextlistErreur[	226	]	 := ;
TextlistErreur[	227	]	 := ;
TextlistErreur[	228	]	 := ;
TextlistErreur[	229	]	 := ;
TextlistErreur[	230	]	 := ;
TextlistErreur[	231	]	 := ;
TextlistErreur[	232	]	 := ;
TextlistErreur[	233	]	 := ;
TextlistErreur[	234	]	 := ;
TextlistErreur[	235	]	 := ;
TextlistErreur[	236	]	 := ;
TextlistErreur[	237	]	 := ;
TextlistErreur[	238	]	 := ;
TextlistErreur[	239	]	 := ;
TextlistErreur[	240	]	 := ;
TextlistErreur[	241	]	 := ;
TextlistErreur[	242	]	 := ;
TextlistErreur[	243	]	 := ;
TextlistErreur[	244	]	 := ;
TextlistErreur[	245	]	 := ;
TextlistErreur[	246	]	 := ;
TextlistErreur[	247	]	 := ;
TextlistErreur[	248	]	 := ;
TextlistErreur[	249	]	 := ;
*)

//warning : 

TextlistErreur[	250	]	 := WarningCarter;
TextlistErreur[	251	]	 := WarningAir;

(*
TextlistErreur[	252	]	 := ;
TextlistErreur[	253	]	 := ;
TextlistErreur[	254	]	 := ;
TextlistErreur[	255	]	 := ;
TextlistErreur[	256	]	 := ;
TextlistErreur[	257	]	 := ;
TextlistErreur[	258	]	 := ;
TextlistErreur[	259	]	 := ;
TextlistErreur[	260	]	 := ;
TextlistErreur[	261	]	 := ;
TextlistErreur[	262	]	 := ;
TextlistErreur[	263	]	 := ;
TextlistErreur[	264	]	 := ;
TextlistErreur[	265	]	 := ;
TextlistErreur[	266	]	 := ;
TextlistErreur[	267	]	 := ;
TextlistErreur[	268	]	 := ;
TextlistErreur[	269	]	 := ;
TextlistErreur[	270	]	 := ;
TextlistErreur[	271	]	 := ;
TextlistErreur[	272	]	 := ;
TextlistErreur[	273	]	 := ;
TextlistErreur[	274	]	 := ;
TextlistErreur[	275	]	 := ;
TextlistErreur[	276	]	 := ;
TextlistErreur[	277	]	 := ;
TextlistErreur[	278	]	 := ;
TextlistErreur[	279	]	 := ;
TextlistErreur[	280	]	 := ;
TextlistErreur[	281	]	 := ;
TextlistErreur[	282	]	 := ;
TextlistErreur[	283	]	 := ;
TextlistErreur[	284	]	 := ;
TextlistErreur[	285	]	 := ;
TextlistErreur[	286	]	 := ;
TextlistErreur[	287	]	 := ;
TextlistErreur[	288	]	 := ;
TextlistErreur[	289	]	 := ;
TextlistErreur[	290	]	 := ;
TextlistErreur[	291	]	 := ;
TextlistErreur[	292	]	 := ;
TextlistErreur[	293	]	 := ;
TextlistErreur[	294	]	 := ;
TextlistErreur[	295	]	 := ;
TextlistErreur[	296	]	 := ;
TextlistErreur[	297	]	 := ;
TextlistErreur[	298	]	 := ;
TextlistErreur[	299	]	 := ;
TextlistErreur[	300	]	 := ;
TextlistErreur[	301	]	 := ;
TextlistErreur[	302	]	 := ;
TextlistErreur[	303	]	 := ;
TextlistErreur[	304	]	 := ;
TextlistErreur[	305	]	 := ;
TextlistErreur[	306	]	 := ;
TextlistErreur[	307	]	 := ;
TextlistErreur[	308	]	 := ;
TextlistErreur[	309	]	 := ;
TextlistErreur[	310	]	 := ;
TextlistErreur[	311	]	 := ;
TextlistErreur[	312	]	 := ;
TextlistErreur[	313	]	 := ;
TextlistErreur[	314	]	 := ;
TextlistErreur[	315	]	 := ;
TextlistErreur[	316	]	 := ;
TextlistErreur[	317	]	 := ;
TextlistErreur[	318	]	 := ;
TextlistErreur[	319	]	 := ;
TextlistErreur[	320	]	 := ;
TextlistErreur[	321	]	 := ;
TextlistErreur[	322	]	 := ;
TextlistErreur[	323	]	 := ;
TextlistErreur[	324	]	 := ;
TextlistErreur[	325	]	 := ;
TextlistErreur[	326	]	 := ;
TextlistErreur[	327	]	 := ;
TextlistErreur[	328	]	 := ;
TextlistErreur[	329	]	 := ;
TextlistErreur[	330	]	 := ;
TextlistErreur[	331	]	 := ;
TextlistErreur[	332	]	 := ;
TextlistErreur[	333	]	 := ;
TextlistErreur[	334	]	 := ;
TextlistErreur[	335	]	 := ;
TextlistErreur[	336	]	 := ;
TextlistErreur[	337	]	 := ;
TextlistErreur[	338	]	 := ;
TextlistErreur[	339	]	 := ;
TextlistErreur[	340	]	 := ;
TextlistErreur[	341	]	 := ;
TextlistErreur[	342	]	 := ;
TextlistErreur[	343	]	 := ;
TextlistErreur[	344	]	 := ;
TextlistErreur[	345	]	 := ;
TextlistErreur[	346	]	 := ;
TextlistErreur[	347	]	 := ;
TextlistErreur[	348	]	 := ;
TextlistErreur[	349	]	 := ;
TextlistErreur[	350	]	 := ;
TextlistErreur[	351	]	 := ;
TextlistErreur[	352	]	 := ;
TextlistErreur[	353	]	 := ;
TextlistErreur[	354	]	 := ;
TextlistErreur[	355	]	 := ;
TextlistErreur[	356	]	 := ;
TextlistErreur[	357	]	 := ;
TextlistErreur[	358	]	 := ;
TextlistErreur[	359	]	 := ;
TextlistErreur[	360	]	 := ;
TextlistErreur[	361	]	 := ;
TextlistErreur[	362	]	 := ;
TextlistErreur[	363	]	 := ;
TextlistErreur[	364	]	 := ;
TextlistErreur[	365	]	 := ;
TextlistErreur[	366	]	 := ;
TextlistErreur[	367	]	 := ;
TextlistErreur[	368	]	 := ;
TextlistErreur[	369	]	 := ;
TextlistErreur[	370	]	 := ;
TextlistErreur[	371	]	 := ;
TextlistErreur[	372	]	 := ;
TextlistErreur[	373	]	 := ;
TextlistErreur[	374	]	 := ;
*)

//warnings toujours acquittables:

TextlistErreur[	375	]	 := WarningMaintenance;
TextlistErreur[	376	]	 := WarningImprimante;

(*
TextlistErreur[	377	]	 := ;
TextlistErreur[	378	]	 := ;
TextlistErreur[	379	]	 := ;
TextlistErreur[	380	]	 := ;
TextlistErreur[	381	]	 := ;
TextlistErreur[	382	]	 := ;
TextlistErreur[	383	]	 := ;
TextlistErreur[	384	]	 := ;
TextlistErreur[	385	]	 := ;
TextlistErreur[	386	]	 := ;
TextlistErreur[	387	]	 := ;
TextlistErreur[	388	]	 := ;
TextlistErreur[	389	]	 := ;
TextlistErreur[	390	]	 := ;
TextlistErreur[	391	]	 := ;
TextlistErreur[	392	]	 := ;
TextlistErreur[	393	]	 := ;
TextlistErreur[	394	]	 := ;
TextlistErreur[	395	]	 := ;
TextlistErreur[	396	]	 := ;
TextlistErreur[	397	]	 := ;
TextlistErreur[	398	]	 := ;
TextlistErreur[	399	]	 := ;
TextlistErreur[	400	]	 := ;
TextlistErreur[	401	]	 := ;
TextlistErreur[	402	]	 := ;
TextlistErreur[	403	]	 := ;
TextlistErreur[	404	]	 := ;
TextlistErreur[	405	]	 := ;
TextlistErreur[	406	]	 := ;
TextlistErreur[	407	]	 := ;
TextlistErreur[	408	]	 := ;
TextlistErreur[	409	]	 := ;
TextlistErreur[	410	]	 := ;
TextlistErreur[	411	]	 := ;
TextlistErreur[	412	]	 := ;
TextlistErreur[	413	]	 := ;
TextlistErreur[	414	]	 := ;
TextlistErreur[	415	]	 := ;
TextlistErreur[	416	]	 := ;
TextlistErreur[	417	]	 := ;
TextlistErreur[	418	]	 := ;
TextlistErreur[	419	]	 := ;
TextlistErreur[	420	]	 := ;
TextlistErreur[	421	]	 := ;
TextlistErreur[	422	]	 := ;
TextlistErreur[	423	]	 := ;
TextlistErreur[	424	]	 := ;
TextlistErreur[	425	]	 := ;
TextlistErreur[	426	]	 := ;
TextlistErreur[	427	]	 := ;
TextlistErreur[	428	]	 := ;
TextlistErreur[	429	]	 := ;
TextlistErreur[	430	]	 := ;
TextlistErreur[	431	]	 := ;
TextlistErreur[	432	]	 := ;
TextlistErreur[	433	]	 := ;
TextlistErreur[	434	]	 := ;
TextlistErreur[	435	]	 := ;
TextlistErreur[	436	]	 := ;
TextlistErreur[	437	]	 := ;
TextlistErreur[	438	]	 := ;
TextlistErreur[	439	]	 := ;
TextlistErreur[	440	]	 := ;
TextlistErreur[	441	]	 := ;
TextlistErreur[	442	]	 := ;
TextlistErreur[	443	]	 := ;
TextlistErreur[	444	]	 := ;
TextlistErreur[	445	]	 := ;
TextlistErreur[	446	]	 := ;
TextlistErreur[	447	]	 := ;
TextlistErreur[	448	]	 := ;
TextlistErreur[	449	]	 := ;
TextlistErreur[	450	]	 := ;
TextlistErreur[	451	]	 := ;
TextlistErreur[	452	]	 := ;
TextlistErreur[	453	]	 := ;
TextlistErreur[	454	]	 := ;
TextlistErreur[	455	]	 := ;
TextlistErreur[	456	]	 := ;
TextlistErreur[	457	]	 := ;
TextlistErreur[	458	]	 := ;
TextlistErreur[	459	]	 := ;
TextlistErreur[	460	]	 := ;
TextlistErreur[	461	]	 := ;
TextlistErreur[	462	]	 := ;
TextlistErreur[	463	]	 := ;
TextlistErreur[	464	]	 := ;
TextlistErreur[	465	]	 := ;
TextlistErreur[	466	]	 := ;
TextlistErreur[	467	]	 := ;
TextlistErreur[	468	]	 := ;
TextlistErreur[	469	]	 := ;
TextlistErreur[	470	]	 := ;
TextlistErreur[	471	]	 := ;
TextlistErreur[	472	]	 := ;
TextlistErreur[	473	]	 := ;
TextlistErreur[	474	]	 := ;
TextlistErreur[	475	]	 := ;
TextlistErreur[	476	]	 := ;
TextlistErreur[	477	]	 := ;
TextlistErreur[	478	]	 := ;
TextlistErreur[	479	]	 := ;
TextlistErreur[	480	]	 := ;
TextlistErreur[	481	]	 := ;
TextlistErreur[	482	]	 := ;
TextlistErreur[	483	]	 := ;
TextlistErreur[	484	]	 := ;
TextlistErreur[	485	]	 := ;
TextlistErreur[	486	]	 := ;
TextlistErreur[	487	]	 := ;
TextlistErreur[	488	]	 := ;
TextlistErreur[	489	]	 := ;
TextlistErreur[	490	]	 := ;
TextlistErreur[	491	]	 := ;
TextlistErreur[	492	]	 := ;
TextlistErreur[	493	]	 := ;
TextlistErreur[	494	]	 := ;
TextlistErreur[	495	]	 := ;
TextlistErreur[	496	]	 := ;
TextlistErreur[	497	]	 := ;
TextlistErreur[	498	]	 := ;
TextlistErreur[	499	]	 := ;
*)
END_ACTION

END_PROGRAM

// ---- GlobalTextList.TcGTLO
TEXTLIST GlobalTextList
  238 = '   Maintenance' | En: '   Maintenance'
  661 = '%.0f' | En: '%.0f'
  215 = '%.0f ' | En: '%.0f'
  648 = '%.0f /' | En: '%.0f /'
  1018 = '%.0f heure(s)' | En: '%.0f hour(s)'
  1709 = '%.0f hrs' | En: '%.0f hrs'
  1058 = '%.0f min' | En: '%.0f min'
  528 = '%.0f minute(s)' | En: '%.0f minute(s)'
  48 = '%.0f sec' | En: '%.0f sec'
  13 = '%.0f seconde(s)' | En: '%.0f second(s)'
  513 = '%.0f Vol/h' | En: '%.0f Vol/h'
  748 = '%.0f °C' | En: '%.0f °C'
  97 = '%.1f L' | En: '%.1f L'
  943 = '%d' | En: '%d'
  52 = '%s' | En: '%s'
  160 = '- Douchette alimentée' | En: '- Handspray supply'
  584 = '- Vidange(s) ouverte(s)' | En: '- Drain(s) opened'
  174 = 'Admin' | En: 'Admin'
  997 = 'Air : %.0f Vol/h' | En: 'Air : %0f Vol/h'
  56 = 'Air : %.1f Vol/h' | En: 'Air : %.1f Vol/h'
  636 = 'ALERTE NIVEAU HAUT BAC A DOUCHE' | En: 'HIGH WATER LEVEL IN SHOWER TRAY ALERT'
  1381 = 'Appli : %.0f %%' | En: 'Apply : %.0f %%'
  1516 = 'Appli : %.0f m3/h' | En: 'Apply : %.0f m3/h'
  10 = "APPUYER SUR LA DOUCHETTE POUR L'UTILISER !" | En: '- PUSH ON HANDSPRAY TO USE IT !'
  305 = 'APPUYER SUR LE BOUTON REARMEMENT' | En: 'PUSH THE REARM BUTTON TO CONTINUE'
  1147 = 'Blow Temp : %.1f °C'
  882 = 'Bow Temp : %.1f °C'
  292 = 'Cabine' | En: 'Booth'
  491 = 'CABINE EN PAUSE' | En: 'BOOTH ON PAUSE'
  99 = 'Chasse WC gros volume' | En: 'Large-volume flush toilet'
  158 = 'Chasse WC petit volume' | En: 'Low-volume flush toilet'
  772 = 'Chasse(s) restante(s) :' | En: 'Remaining flush(s) :'
  31 = 'CHWS Temp : %.1f °C'
  1236 = 'COM Registre soufflage' | En: 'Supply air damper com.'
  230 = 'Connecté' | En: 'Connected'
  619 = 'Connexion' | En: 'Connection'
  912 = 'Cons. Hygro. : %.1f %%Hr' | En: 'Set. Hygro. : %.1f %%Hr'
  225 = 'Cons. Temp. : %.1f °C' | En: 'Set. Temp. : %.1f °C'
  1388 = 'Cons. Temp. eau : %.1f °C' | En: 'Set. Temp. Wat. : %.1f °C'
  117 = 'Consigne : %.0f Vol/h' | En: 'Setpoint : %.0f Vol/h'
  340 = 'Consigne : %.1f L' | En: 'Setpoint : %.1f L'
  894 = 'Consigne(s) : %.1f L' | En: 'Setpoint : %.1f L'
  886 = 'Contact' | En: 'Contact'
  458 = 'Debit Max : %d Vol/h' | En: 'Flow max : %d Vol/h'
  195 = 'Debit Min : %d Vol/h' | En: 'Flow min : %d Vol/h'
  734 = 'Deconnecté' | En: 'Disconnected'
  821 = 'Deconnexion' | En: 'Deconnection'
  255 = 'Depollution' | En: 'Decontamination'
  975 = 'Douchette' | En: 'Hand Spray'
  617 = 'Drain douche' | En: 'Shower drain'
  469 = 'Drain lavabo' | En: 'Sink drain'
  784 = 'Débit : %.1f l/min' | En: 'Flow : %.1f l/min'
  1121 = 'Débit : %d m3/h' | En: 'Flow : %d m3/h'
  1233 = 'Défaut différentiel prise électrique' | En: 'Differential fault in electrical outlet'
  478 = 'Défaut discordance débit d’eau de la douche' | En: 'Mismatch in shower water flow rate'
  799 = 'Défaut discordance débit d’eau du lavabo' | En: 'Mismatch in sink water flow rate'
  633 = 'Défaut discordance prise de courant' | En: 'Power plug supply mismatch'
  514 = 'Défaut prise forcée manuellement' | En: 'Manually forced power plug'
  1537 = 'Défaut prise lors de l’ouverture porte' | En: 'Door open during a power plug cycle'
  801 = 'Défaut temperature de soufflage CTA climatique trop haute' | En: 'Faulty supply air temperature AHU climatic too high'
  586 = 'Détail de la recette sélectionnée' | En: 'Details of the selected protocol'
  1156 = 'Eau : %.1f °C' | En: 'Wat : %.1f °C'
  1560 = 'Ecr paramètres' | En: 'Wrt Settings'
  844 = 'Electrovanne douche' | En: 'Shower solenoid valve'
  684 = 'Electrovanne lavabo' | En: 'Sink solenoid valve'
  415 = 'Etape : %d /' | En: 'Step : %d /'
  318 = 'Etats des E/S TOR' | En: 'States of I/O'
  1440 = 'ETOR10_Hygrostat_Souf_CT'
  1495 = 'ETOR11_Pressostat_Secu'
  1076 = 'ETOR12_Thermostat_Secu'
  493 = 'ETOR13_Marche_BatElec_CTA'
  273 = 'ETOR1_Fdc_Va_Vid_Lavabo_Ouv'
  949 = 'ETOR2_Fdc_Va_Vid_Lavabo_Ferm'
  1342 = 'ETOR3_Info_Ma_Prise'
  829 = 'ETOR3_Reg_BasDebit_Souf_Ouv'
  1108 = 'ETOR4_RegBasDebit_Souf_Ferm'
  1346 = 'ETOR4_Service_Humi_CTA'
  275 = 'ETOR5_Def_Humi_CTA'
  82 = 'ETOR5_Reg_BasDebit_Ext_Ouv'
  892 = 'ETOR6_Info_Contact_Porte'
  1455 = 'ETOR6_Reg_BasDebit_Ext_Ferm'
  926 = 'ETOR7_Def_MotRep_Souf_CTA'
  1403 = 'ETOR7_Info_Ma_Prise'
  258 = 'ETOR8_Def_MotSouf_Souf_CTA'
  401 = 'ETOR8_Info_Contact_Porte'
  1031 = 'ETOR9_Def_Alim_BatElec_CTA'
  665 = 'EXTRACTION' | En: 'EXHAUST'
  566 = 'Extraction' | En: 'Exhaust'
  164 = 'Extraction bas débit' | En: 'Low- flow exhaust'
  519 = 'FDC :' | En: 'LS'
  168 = 'FERM' | En: 'CLS'
  279 = 'Fermer' | En: 'Closed'
  779 = 'Fermé' | En: 'Close'
  773 = 'FORCE' | En: 'FORCE'
  223 = 'Heure(s) :' | En: 'Hour(s) :'
  670 = 'Heure(s) restante(s) :' | En: 'Remaining hour(s) :'
  936 = 'Hygro : %.1f %Hr' | En: 'Hygro : %.1f %Hr'
  126 = 'LED' | En: 'LED'
  1475 = 'Mail : Smartbooth@osmose06.com' | En: 'Mail : Smartbooth@osmose06.com'
  581 = 'Mesure : %.0f %%' | En: 'Measure : %.0f %%'
  434 = 'Mesure : %.0f m3/h' | En: 'Measure : %.0f m3/h'
  1096 = 'Mesure : %.0f Vol/h' | En: 'Measure : %.0f Vol/h'
  887 = 'Minute(s) :' | En: 'Minute(s) :'
  797 = 'Minute(s) restante(s) :' | En: 'Remaining minute(s) :'
  354 = 'MODE' | En: 'MODE'
  885 = 'MODE DEPOLLUTION EN COURS' | En: 'DECONTAMINATION IN PROGRESS'
  346 = 'Mode maintenance' | En: 'Maintenance mode'
  977 = 'Mode manuel' | En: 'Manual mode'
  976 = 'MODE MANUEL EN COURS' | En: 'MANUAL MODE IN PROGRESS'
  920 = 'MODE NETTOYAGE EN COURS' | En: 'CLEANING IN PROGRES'
  1032 = 'Mode N°%.0f' | En: 'Mode N°%.0f'
  718 = 'Mode N°%d' | En: 'Mode N°%d'
  432 = 'MODE RECETTE EN COURS' | En: 'PROTOCOL IN PROGRES'
  224 = 'Moteur bas débit' | En: 'Low-flow motor'
  685 = 'Moteur reprise' | En: 'Exhaust motor'
  789 = 'Moteur soufflage' | En: 'Supply motor'
  878 = 'Nbre chasse :' | En: 'Nber Flush :'
  911 = 'Next' | En: 'Next'
  923 = 'None' | En: 'None'
  41 = 'NORMAL' | En: 'NORMAL'
  585 = 'Off' | En: 'Off'
  88 = 'On' | En: 'On'
  565 = 'Operator' | En: 'Operator'
  157 = 'OUT' | En: 'OUT'
  860 = 'OUV' | En: 'OPN'
  395 = 'Ouvert' | En: 'Open'
  1034 = 'Ouverture : %.0f %%' | En: 'Opening : %.0f %%'
  113 = 'Pause' | En: 'Pause'
  649 = 'Phone : +33 (0)4 93 77 79 74' | En: 'Phone : +33 (0)4 93 77 79 74'
  1155 = 'Position : %.0f %%' | En: 'Position : %.0f %%'
  1383 = 'Press : %.0f Pa' | En: 'Press : %.0f Pa'
  1439 = 'Press Ext : %.0f Pa' | En: 'Ext Press : %.0f Pa'
  690 = 'Press Souf : %.0f Pa' | En: 'Spl Press : %.0f Pa'
  934 = 'Prise électrique' | En: 'Electrical outlet'
  687 = 'Re-Start' | En: 'Re-Start'
  964 = 'Recettes' | En: 'Protocols'
  877 = 'Retour' | En: 'Return'
  891 = 'Réarmement' | En: 'Rearm'
  712 = 'Réarmer' | En: 'Rearm'
  573 = 'Seconde(s) :' | En: 'Second(s) :'
  688 = 'Seconde(s) restante(s) :' | En: 'Remaining second(s) :'
  369 = 'Service' | En: 'Service'
  924 = 'SOUFFLAGE' | En: 'SUPPLY'
  69 = 'Soufflage' | En: 'Supply'
  249 = 'Soufflage bas débit' | En: 'Low-Flow supply'
  626 = 'Start' | En: 'Start'
  246 = 'Stop' | En: 'Stop'
  1079 = 'STOR1_Cmd_EV_Alim_Lavabo'
  1180 = 'STOR1_Cmd_Va_Vid_Lavabo'
  747 = 'STOR2_Cmd_EV_Alim_Lavabo'
  284 = 'STOR2_Cmd_Va_Vid_Lavabo'
  4 = 'STOR3_Cmd_Ma_Prise'
  1277 = 'STOR3_Cmd_Reg_BasDebit_Souf'
  837 = 'STOR4_Cmd_BatElec_CTA'
  1340 = 'STOR4_Cmd_Reg_BasDebit_Ext'
  867 = 'STOR5_Cmd_Ma_Prise'
  488 = 'Suivant' | En: 'Next'
  196 = 'Temp : %.1f °C' | En: 'Temp : %.1f °C'
  525 = 'Temp. eau :' | En: 'Temp. Wat. :'
  319 = 'Validation' | En: 'Validation'
  544 = 'Vanne Bat. froide' | En: 'Cold Bat. valve'
  435 = 'Vanne douche' | En: 'Shower valve'
  548 = 'Vanne eau mitigée' | En: 'Mixed water valve'
  763 = 'Vanne lavabo' | En: 'Sink valve'
  506 = 'Vanne NEP' | En: 'CIP valve'
  543 = 'Ventilation :' | En: 'Ventilation :'
  307 = 'Veuillez sélectionner une recette' | En: 'Please select a protocol'
  1396 = 'Vit Max : %.0f %%' | En: 'Max spd : %.0f %%'
  1419 = 'Vit Min : %.0f %%' | En: 'Min spd : %.0f %%'
  108 = 'Vitesse : %.0f %%' | En: 'Speed : %.0f %%'
  363 = "Vol. d'eau :" | En: 'Wat. vol. :'
  735 = "Volume d'eau : %.1f L" | En: 'Water Flow : %.1f L'
END_TEXTLIST

// ---- Visualizations/Visualizations/Accueil.TcVIS
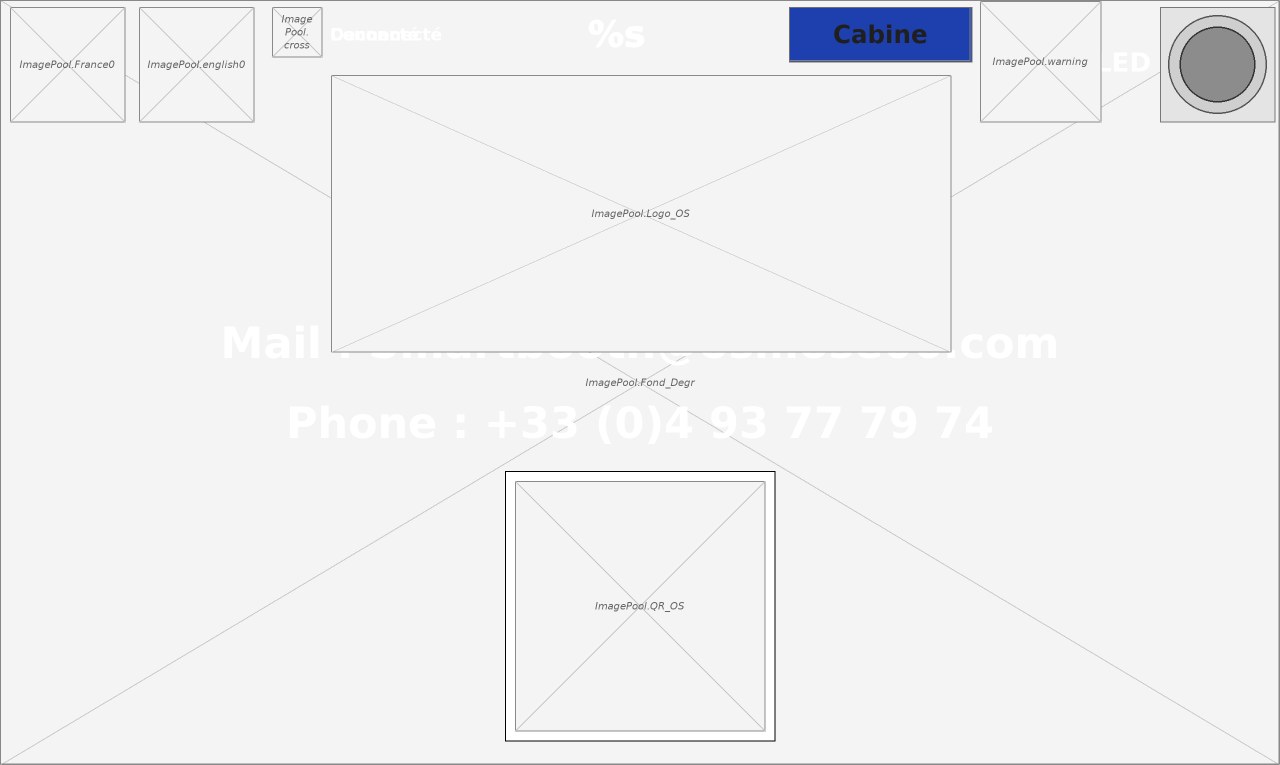
VISUALIZATION Accueil  // 1280x765
    Frame (0,0 1280x765)
        shows masque()
    RoundedRectangle (0,383 1280x80), "Phone : +33 (0)4 93 77 79 74"
    RoundedRectangle (0,303 1280x80), "Mail : Smartbooth@osmose06.com"
    RoundedRectangle (340,153 600x126)
    Image (331,75 620x277), image: ImagePool.Logo_OS
    Rectangle (0,128 1278x633)
        OnMouseDown: change screen: menu
    Group (505,471 270x270)
        RoundedRectangle (0,0 270x270)
        Image (10,10 250x250), image: ImagePool.QR_OS
END_VISUALIZATION

// ---- Visualizations/Visualizations/Depollution.TcVIS
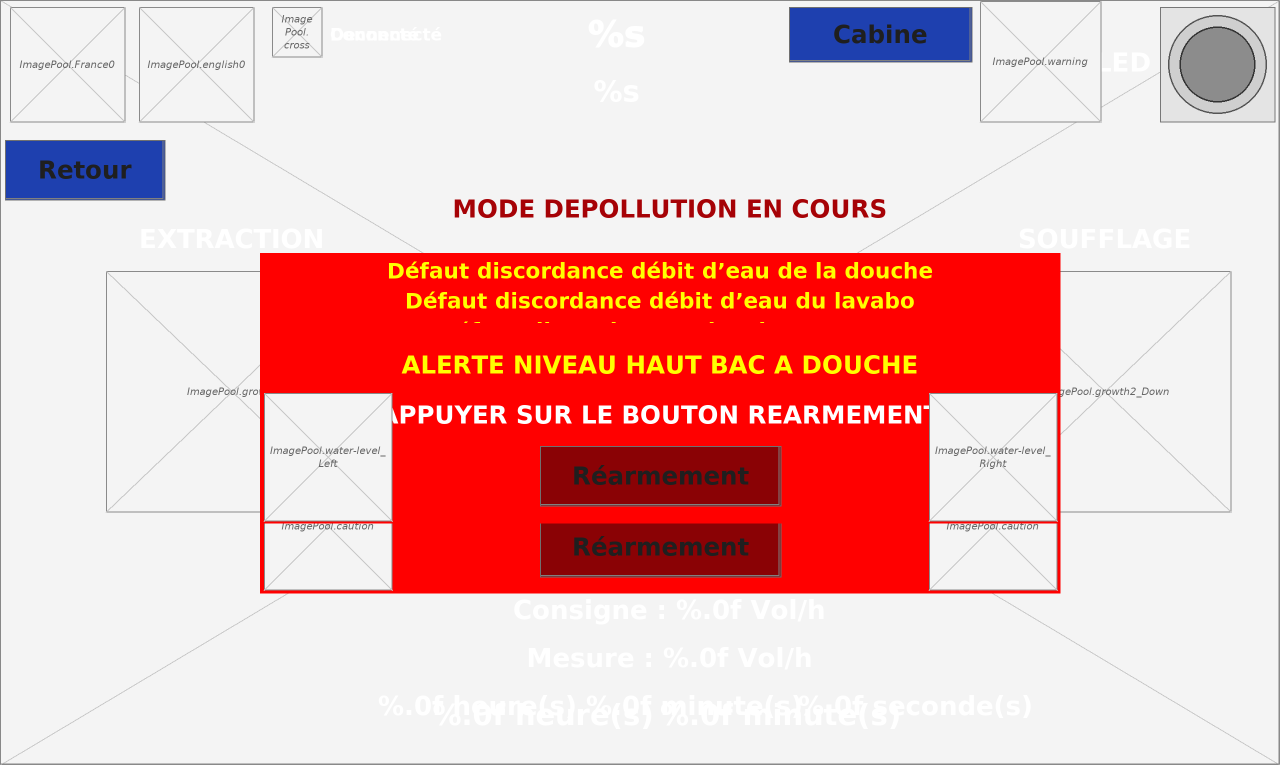
VISUALIZATION Depollution  // 1280x765
    Frame (0,0 1280x765)
        shows masque()
    Button (5,140 160x60), "Retour", invisible if: Mode_Cabine_Depollution
        OnMouseDown: change screen: menu
    Image (501,255 322x322), image: ImagePool_Buttons.Button_Appuie_Sombre
    Image (501,255 322x322), invisible if: Start_Etat_Depollution, image: ImagePool_Buttons.Button_NonAppuie_Sombre
        OnMouseDown: toggle Start_Etat_Depollution
    Image (106,271 252x241), image: ImagePool.growth
        p2738717112: GVL_Visu.Arrow_Up
    Image (979,271 252x241), image: ImagePool.growth2_Down
        p2738717112: GVL_Visu.Arrow_Down
    Rectangle (106,214 252x50), "EXTRACTION"
    Rectangle (979,214 252x50), "SOUFFLAGE"
    Group (265,185 809x545), invisible if: NOT Mode_Cabine_Depollution
        Rectangle (81,0 648x48), "MODE DEPOLLUTION EN COURS", invisible if: GVL_Visu.On_Off_Anim
        Group (0,497 809x48)
            Rectangle (0,0 315x48), "%.0f heure(s)", text variable: Lect_Temp_heure_Depol, invisible if: NOT Mode_Cabine_Depollution
            Rectangle (318,0 220x48), "%.0f minute(s)", text variable: Lect_Temp_Minute_Depol, invisible if: NOT Mode_Cabine_Depollution
            Rectangle (530,0 279x48), "%.0f seconde(s)", text variable: Lect_Temp_Seconde_Depol, invisible if: NOT Mode_Cabine_Depollution
    Rectangle (444,586 451x48), "Consigne : %.0f Vol/h", text variable: Cons_Deb_Souf_Etat_Depol
    Rectangle (444,634 451x48), "Mesure : %.0f Vol/h", text variable: Visu.IHM_Mesure_Debit_Deconta
    Group (420,683 500x64), invisible if: Mode_Cabine_Depollution
        RoundedRectangle (0,0 237x64), "%.0f heure(s)", text variable: Cons_Temp_heure_Depol
            OnMouseDown: write the text variable via VisuDialogs.Numpad, min 0, max 23, format %.0f
        RoundedRectangle (237,0 263x64), "%.0f minute(s)", text variable: Cons_Temp_Minute_Depol
            OnMouseDown: write the text variable via VisuDialogs.Numpad, min 0, max 59, format %.0f
    Group (260,253 800x340)
        Frame (0,0 800x340), invisible if: NOT GVL_Visu.Affichage_PopUp_Alarm
            shows PopUp_Alarms()
        Frame (0,70 800x200), invisible if: NOT GVL_Visu.Affichage_PopUp_HightLevel
            shows PopUp_Hight_Level()
END_VISUALIZATION

// ---- Visualizations/Visualizations/Fonds/masque.TcVIS
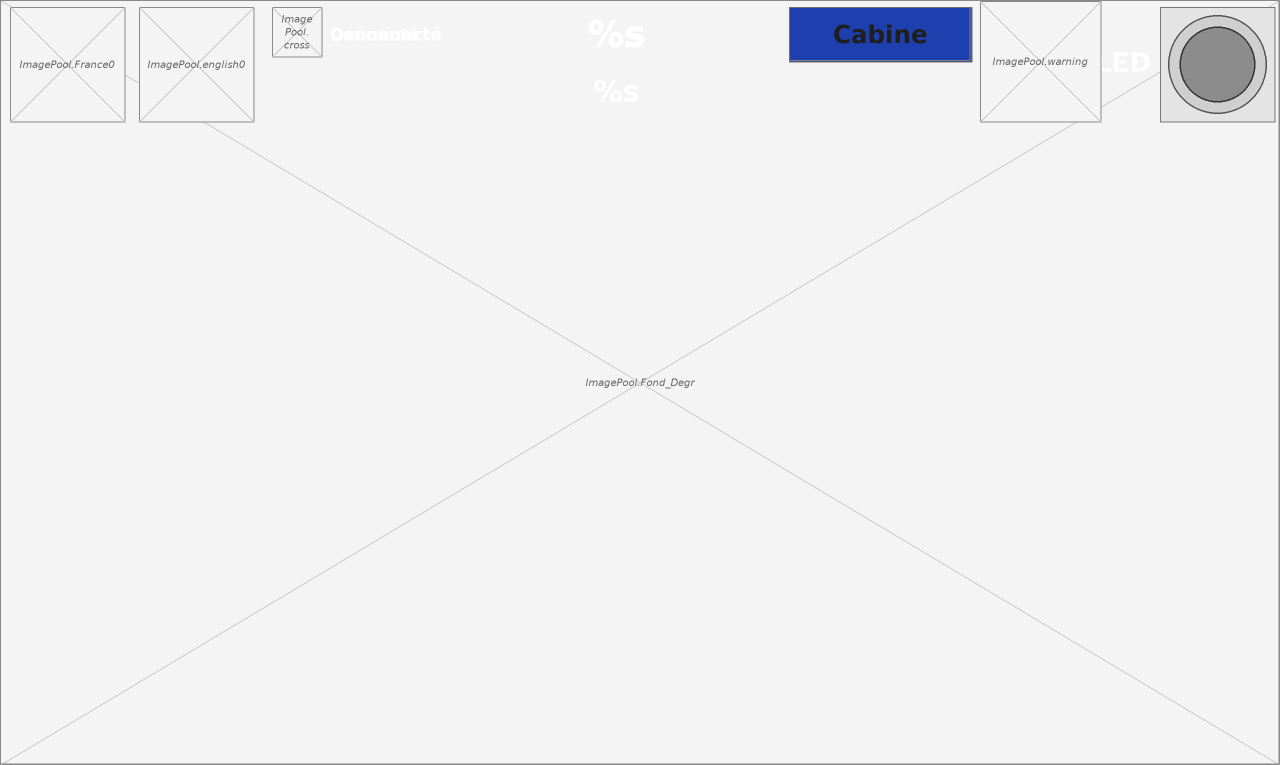
VISUALIZATION masque  // 1280x765
    Image (0,0 1280x765), image: ImagePool.Fond_Degr
    PushSwitch (1160,7 115x115), variable: Activation_Ecl, behaviour: TOGGLE, style: Switch-PushSwitch-Gray
    Image (10,7 115x115), image: ImagePool.France0
        OnMouseDown: ChangeLanguage ChangeLanguage=fr
    Image (139,7 115x115), image: ImagePool.english0
        OnMouseDown: ChangeLanguage ChangeLanguage=En
    Rectangle (262,64 710x55), "%s", text list: 'Etats_Cabine', text index: Sel_Etats_Cabine
        p55702900: GVL_Visu.Couleur_Cabine2
    Rectangle (463,7 309x53), "%s", text variable: GVL_Visu.Nom_Cabine_EN, invisible if: VisuElems.CURRENTLANGUAGE = 'fr'
    Group (272,7 196x53)
        Image (0,0 50x50), image: ImagePool.checked
        Image (0,0 50x50), invisible if: GVL_Visu.Etat_Connexion, image: ImagePool.cross
        Rectangle (55,0 141x55), "Deconnecté", invisible if: GVL_Visu.Etat_Connexion
        Rectangle (55,0 141x55), "Connecté"
    Rectangle (463,7 307x55), "%s", text variable: GVL_Visu.Nom_Cabine_FR, invisible if: VisuElems.CURRENTLANGUAGE = 'en'
    Rectangle (1073,36 81x53), "LED"
    Button (789,7 183x55), "Cabine"
        OnMouseDown: OpenDialog Dialog=Actionneurs, OpenModal=True, PositionX=0, PositionY=0
    Group (980,1 121x121)
        Image (2,4 113x113), invisible if: GVL_Visu.On_Off_Anim_Lent OR NOT Mode_Warning, image: ImagePool.caution
            OnMouseDown: OpenDialog Dialog=Alarmes, OpenModal=True, PositionX=0, PositionY=0
        Image (0,0 121x121), invisible if: GVL_Visu.On_Off_Anim_Lent OR NOT Mode_Cabine_Defaut, image: ImagePool.warning
            OnMouseDown: OpenDialog Dialog=Alarmes, OpenModal=True, PositionX=0, PositionY=0
END_VISUALIZATION

